   (*считывание и обработка дискретного сигнала с выбранного канала*)
   CASE #N_module OF
       4:  // Модуль 4
           CASE #N_chanel OF
               1:  #Signal := "Module4Chanel1";   //Канал 1
               2:  #Signal := "Module4Chanel2";   //Канал 2
               3:  #Signal := "Module4Chanel3";   //Канал 3
               4:  #Signal := "Module4Chanel4";   //Канал 4
               5:  #Signal := "Module4Chanel5";   //Канал 5
               6:  #Signal := "Module4Chanel6";   //Канал 6
               7:  #Signal := "Module4Chanel7";   //Канал 7
               8:  #Signal := "Module4Chanel8";   //Канал 8
               9:  #Signal := "Module4Chanel9";   //Канал 9
               10: #Signal := "Module4Chanel10";  //Канал 10
               11: #Signal := "Module4Chanel11";  //Канал 11
               12: #Signal := "Module4Chanel12";  //Канал 12
               13: #Signal := "Module4Chanel13";  //Канал 13
               14: #Signal := "Module4Chanel14";  //Канал 14
               15: #Signal := "Module4Chanel15";  //Канал 15
               16: #Signal := "Module4Chanel16";  //Канал 16
               ELSE
                   #Signal := FALSE;
           END_CASE;
       5:  // Модуль 5
           CASE #N_chanel OF
               1:  #Signal := "Module5Chanel1";   //Канал 1
               2:  #Signal := "Module5Chanel2";   //Канал 2
               3:  #Signal := "Module5Chanel3";   //Канал 3
               4:  #Signal := "Module5Chanel4";   //Канал 4
               5:  #Signal := "Module5Chanel5";   //Канал 5
               6:  #Signal := "Module5Chanel6";   //Канал 6
               7:  #Signal := "Module5Chanel7";   //Канал 7
               8:  #Signal := "Module5Chanel8";   //Канал 8
               9:  #Signal := "Module5Chanel9";   //Канал 9
               10: #Signal := "Module5Chanel10";  //Канал 10
               11: #Signal := "Module5Chanel11";  //Канал 11
               12: #Signal := "Module5Chanel12";  //Канал 12
               13: #Signal := "Module5Chanel13";  //Канал 13
               14: #Signal := "Module5Chanel14";  //Канал 14
               15: #Signal := "Module5Chanel15";  //Канал 15
               16: #Signal := "Module5Chanel16";  //Канал 16
               ELSE
                   #Signal := FALSE;
           END_CASE;
       6:  // Модуль 6
           CASE #N_chanel OF
               1:  #Signal := "Module6Chanel1";   //Канал 1
               2:  #Signal := "Module6Chanel2";   //Канал 2
               3:  #Signal := "Module6Chanel3";   //Канал 3
               4:  #Signal := "Module6Chanel4";   //Канал 4
               5:  #Signal := "Module6Chanel5";   //Канал 5
               6:  #Signal := "Module6Chanel6";   //Канал 6
               7:  #Signal := "Module6Chanel7";   //Канал 7
               8:  #Signal := "Module6Chanel8";   //Канал 8
               9:  #Signal := "Module6Chanel9";   //Канал 9
               10: #Signal := "Module6Chanel10";  //Канал 10
               11: #Signal := "Module6Chanel11";  //Канал 11
               12: #Signal := "Module6Chanel12";  //Канал 12
               13: #Signal := "Module6Chanel13";  //Канал 13
               14: #Signal := "Module6Chanel14";  //Канал 14
               15: #Signal := "Module6Chanel15";  //Канал 15
               16: #Signal := "Module6Chanel16";  //Канал 16
               ELSE
                   #Signal := FALSE;
           END_CASE;
       7:  // Модуль 7
           CASE #N_chanel OF
               1:  #Signal := "Module7Chanel1";   //Канал 1
               2:  #Signal := "Module7Chanel2";   //Канал 2
               3:  #Signal := "Module7Chanel3";   //Канал 3
               4:  #Signal := "Module7Chanel4";   //Канал 4
               5:  #Signal := "Module7Chanel5";   //Канал 5
               6:  #Signal := "Module7Chanel6";   //Канал 6
               7:  #Signal := "Module7Chanel7";   //Канал 7
               8:  #Signal := "Module7Chanel8";   //Канал 8
               9:  #Signal := "Module7Chanel9";   //Канал 9
               10: #Signal := "Module7Chanel10";  //Канал 10
               11: #Signal := "Module7Chanel11";  //Канал 11
               12: #Signal := "Module7Chanel12";  //Канал 12
               13: #Signal := "Module7Chanel13";  //Канал 13
               14: #Signal := "Module7Chanel14";  //Канал 14
               15: #Signal := "Module7Chanel15";  //Канал 15
               16: #Signal := "Module7Chanel16";  //Канал 16
               ELSE
                   #Signal := FALSE;
           END_CASE;
       8:  // Модуль 8
           CASE #N_chanel OF
               1:  #Signal := "Module8Chanel1";   //Канал 1
               2:  #Signal := "Module8Chanel2";   //Канал 2
               3:  #Signal := "Module8Chanel3";   //Канал 3
               4:  #Signal := "Module8Chanel4";   //Канал 4
               5:  #Signal := "Module8Chanel5";   //Канал 5
               6:  #Signal := "Module8Chanel6";   //Канал 6
               7:  #Signal := "Module8Chanel7";   //Канал 7
               8:  #Signal := "Module8Chanel8";   //Канал 8
               9:  #Signal := "Module8Chanel9";   //Канал 9
               10: #Signal := "Module8Chanel10";  //Канал 10
               11: #Signal := "Module8Chanel11";  //Канал 11
               12: #Signal := "Module8Chanel12";  //Канал 12
               13: #Signal := "Module8Chanel13";  //Канал 13
               14: #Signal := "Module8Chanel14";  //Канал 14
               15: #Signal := "Module8Chanel15";  //Канал 15
               16: #Signal := "Module8Chanel16";  //Канал 16
               ELSE
                   #Signal := FALSE;
           END_CASE;
       9:  // Модуль 9
           CASE #N_chanel OF
               1:  #Signal := "Module9Chanel1";   //Канал 1
               2:  #Signal := "Module9Chanel2";   //Канал 2
               3:  #Signal := "Module9Chanel3";   //Канал 3
               4:  #Signal := "Module9Chanel4";   //Канал 4
               5:  #Signal := "Module9Chanel5";   //Канал 5
               6:  #Signal := "Module9Chanel6";   //Канал 6
               7:  #Signal := "Module9Chanel7";   //Канал 7
               8:  #Signal := "Module9Chanel8";   //Канал 8
               9:  #Signal := "Module9Chanel9";   //Канал 9
               10: #Signal := "Module9Chanel10";  //Канал 10
               11: #Signal := "Module9Chanel11";  //Канал 11
               12: #Signal := "Module9Chanel12";  //Канал 12
               13: #Signal := "Module9Chanel13";  //Канал 13
               14: #Signal := "Module9Chanel14";  //Канал 14
               15: #Signal := "Module9Chanel15";  //Канал 15
               16: #Signal := "Module9Chanel16";  //Канал 16
               ELSE
                   #Signal := FALSE;
           END_CASE;
       ELSE
           #Signal := 0;
   END_CASE;
   IF NOT #Invert THEN
       #Value := #Signal;
   ELSE
       #Value := NOT #Signal;
   END_IF;
END_FUNCTION

FUNCTION "Write_outputs" : Void   // FC4, SCL
{ S7_Optimized_Access := 'TRUE' }
VERSION : 0.1
BEGIN
   (*ЗАПИСЬ ВЫХОДОВ*)
   (*Запись дискретных выходов*)
   (*ЗРГ команда «Больше»*)
   IF "Sensors".ZRG_control_open.Enable THEN
       "Write_discret_signal"(N_module := "Sensors".ZRG_control_open.N_module,
                              N_chanel := "Sensors".ZRG_control_open.N_chanel,
                              Value := "Sensors".ZRG_control_open.Value);
   END_IF;

   (*ЗРГ команда «Меньше»*)
   IF "Sensors".ZRG_control_close.Enable THEN
       "Write_discret_signal"(N_module := "Sensors".ZRG_control_close.N_module,
                              N_chanel := "Sensors".ZRG_control_close.N_chanel,
                              Value := "Sensors".ZRG_control_close.Value);
   END_IF;

   (*НАВ команда «Больше»*)
   IF "Sensors".NAV_control_open.Enable THEN
       "Write_discret_signal"(N_module := "Sensors".NAV_control_open.N_module,
                              N_chanel := "Sensors".NAV_control_open.N_chanel,
                              Value := "Sensors".NAV_control_open.Value);
   END_IF;

   (*НАВ команда «Меньше»*)
   IF "Sensors".NAV_control_close.Enable THEN
       "Write_discret_signal"(N_module := "Sensors".NAV_control_close.N_module,
                              N_chanel := "Sensors".NAV_control_close.N_chanel,
                              Value := "Sensors".NAV_control_close.Value);
   END_IF;

   (*НАД команда «Больше»*)
   IF "Sensors".NAD_control_open.Enable THEN
       "Write_discret_signal"(N_module := "Sensors".NAD_control_open.N_module,
                              N_chanel := "Sensors".NAD_control_open.N_chanel,
                              Value := "Sensors".NAD_control_open.Value);
   END_IF;

   (*НАД команда «Меньше»*)
   IF "Sensors".NAD_control_close.Enable THEN
       "Write_discret_signal"(N_module := "Sensors".NAD_control_close.N_module,
                              N_chanel := "Sensors".NAD_control_close.N_chanel,
                              Value := "Sensors".NAD_control_close.Value);
   END_IF;

   (*Индикация «Работа»*)
   IF "Sensors".Indication_RUN.Enable THEN
       "Write_discret_signal"(N_module := "Sensors".Indication_RUN.N_module,
                              N_chanel := "Sensors".Indication_RUN.N_chanel,
                              Value := "Sensors".Indication_RUN.Value);
   END_IF;

   (*Индикация «Авария»*)
   IF "Sensors".Indication_ALARM.Enable THEN
       "Write_discret_signal"(N_module := "Sensors".Indication_ALARM.N_module,
                              N_chanel := "Sensors".Indication_ALARM.N_chanel,
                              Value := "Sensors".Indication_ALARM.Value);
   END_IF;

   (*Индикация «Защиты в норме»*)
   IF "Sensors".Indication_NORMA.Enable THEN
       "Write_discret_signal"(N_module := "Sensors".Indication_NORMA.N_module,
                              N_chanel := "Sensors".Indication_NORMA.N_chanel,
                              Value := "Sensors".Indication_NORMA.Value);
   END_IF;

   (*Индикация «Готов к розжигу»*)
   IF "Sensors".Indication_READY.Enable THEN
       "Write_discret_signal"(N_module := "Sensors".Indication_READY.N_module,
                              N_chanel := "Sensors".Indication_READY.N_chanel,
                              Value := "Sensors".Indication_READY.Value);
   END_IF;

   (*ЗДГ команда «открыть»*)
   IF "Sensors".ZDG_control_open.Enable THEN
       "Write_discret_signal"(N_module := "Sensors".ZDG_control_open.N_module,
                              N_chanel := "Sensors".ZDG_control_open.N_chanel,
                              Value := "Sensors".ZDG_control_open.Value);
   END_IF;

   (*ЗДГ команда «закрыть»*)
   IF "Sensors".ZDG_control_close.Enable THEN
       "Write_discret_signal"(N_module := "Sensors".ZDG_control_close.N_module,
                              N_chanel := "Sensors".ZDG_control_close.N_chanel,
                              Value := "Sensors".ZDG_control_close.Value);
   END_IF;

   (*ЗДГ команда «стоп»*)
   IF "Sensors".ZDG_control_stop.Enable THEN
       "Write_discret_signal"(N_module := "Sensors".ZDG_control_stop.N_module,
                              N_chanel := "Sensors".ZDG_control_stop.N_chanel,
                              Value := "Sensors".ZDG_control_stop.Value);
   END_IF;

   (*ЗДГ команда «запрет открытия»*)
   IF "Sensors".ZDG_control_disable_open.Enable THEN
       "Write_discret_signal"(N_module := "Sensors".ZDG_control_disable_open.N_module,
                              N_chanel := "Sensors".ZDG_control_disable_open.N_chanel,
                              Value := "Sensors".ZDG_control_disable_open.Value);
   END_IF;

   (*КБ команда «закрыть»*)
   IF "Sensors".KB_control_close.Enable THEN
       "Write_discret_signal"(N_module := "Sensors".KB_control_close.N_module,
                              N_chanel := "Sensors".KB_control_close.N_chanel,
                              Value := "Sensors".KB_control_close.Value);
   END_IF;

   (*КО команда «открыть»*)
   IF "Sensors".KO_control_open.Enable THEN
       "Write_discret_signal"(N_module := "Sensors".KO_control_open.N_module,
                              N_chanel := "Sensors".KO_control_open.N_chanel,
                              Value := "Sensors".KO_control_open.Value);
   END_IF;

   (*КЗ команда «открыть»*)
   IF "Sensors".KZ_control_open.Enable THEN
       "Write_discret_signal"(N_module := "Sensors".KZ_control_open.N_module,
                              N_chanel := "Sensors".KZ_control_open.N_chanel,
                              Value := "Sensors".KZ_control_open.Value);
   END_IF;

   (*ИВН команда «включить»*)
   IF "Sensors".IVN_control_on.Enable THEN
       "Write_discret_signal"(N_module := "Sensors".IVN_control_on.N_module,
                              N_chanel := "Sensors".IVN_control_on.N_chanel,
                              Value := "Sensors".IVN_control_on.Value);
   END_IF;

   (*ПЗК1 команда «открыть»*)
   IF "Sensors".PZK1_control_open.Enable THEN
       "Write_discret_signal"(N_module := "Sensors".PZK1_control_open.N_module,
                              N_chanel := "Sensors".PZK1_control_open.N_chanel,
                              Value := "Sensors".PZK1_control_open.Value);
   END_IF;

   (*ПЗК2 команда «открыть»*)
   IF "Sensors".PZK2_control_open.Enable THEN
       "Write_discret_signal"(N_module := "Sensors".PZK2_control_open.N_module,
                              N_chanel := "Sensors".PZK2_control_open.N_chanel,
                              Value := "Sensors".PZK2_control_open.Value);
   END_IF;

   (*ЗДСВ перед котлом команда «открыть»*)
   IF "Sensors".ZDSV_before_boiler_control_open.Enable THEN
       "Write_discret_signal"(N_module := "Sensors".ZDSV_before_boiler_control_open.N_module,
                              N_chanel := "Sensors".ZDSV_before_boiler_control_open.N_chanel,
                              Value := "Sensors".ZDSV_before_boiler_control_open.Value);
   END_IF;

   (*ЗДСВ перед котлом команда «закрыть»*)
   IF "Sensors".ZDSV_before_boiler_control_close.Enable THEN
       "Write_discret_signal"(N_module := "Sensors".ZDSV_before_boiler_control_close.N_module,
                              N_chanel := "Sensors".ZDSV_before_boiler_control_close.N_chanel,
                              Value := "Sensors".ZDSV_before_boiler_control_close.Value);
   END_IF;

   (*ЗДСВ перед котлом команда «стоп»*)
   IF "Sensors".ZDSV_before_boiler_control_stop.Enable THEN
       "Write_discret_signal"(N_module := "Sensors".ZDSV_before_boiler_control_stop.N_module,
                              N_chanel := "Sensors".ZDSV_before_boiler_control_stop.N_chanel,
                              Value := "Sensors".ZDSV_before_boiler_control_stop.Value);
   END_IF;

   (*ЗДСВ перед котлом команда «разрешение на закрытие»*)
   IF "Sensors".ZDSV_before_boiler_control_disable_close.Enable THEN
       "Write_discret_signal"(N_module := "Sensors".ZDSV_before_boiler_control_disable_close.N_module,
                              N_chanel := "Sensors".ZDSV_before_boiler_control_disable_close.N_chanel,
                              Value := "Sensors".ZDSV_before_boiler_control_disable_close.Value);
   END_IF;

   (*ЗДСВ после котла команда «открыть»*)
   IF "Sensors".ZDSV_after_boiler_control_open.Enable THEN
       "Write_discret_signal"(N_module := "Sensors".ZDSV_after_boiler_control_open.N_module,
                              N_chanel := "Sensors".ZDSV_after_boiler_control_open.N_chanel,
                              Value := "Sensors".ZDSV_after_boiler_control_open.Value);
   END_IF;

   (*ЗДСВ после котла команда «закрыть»*)
   IF "Sensors".ZDSV_after_boiler_control_close.Enable THEN
       "Write_discret_signal"(N_module := "Sensors".ZDSV_after_boiler_control_close.N_module,
                              N_chanel := "Sensors".ZDSV_after_boiler_control_close.N_chanel,
                              Value := "Sensors".ZDSV_after_boiler_control_close.Value);
   END_IF;

   (*ЗДСВ после котла команда «стоп»*)
   IF "Sensors".ZDSV_after_boiler_control_stop.Enable THEN
       "Write_discret_signal"(N_module := "Sensors".ZDSV_after_boiler_control_stop.N_module,
                              N_chanel := "Sensors".ZDSV_after_boiler_control_stop.N_chanel,
                              Value := "Sensors".ZDSV_after_boiler_control_stop.Value);
   END_IF;

   (*ЗДСВ после котла команда «разрешение на закрытие»*)
   IF "Sensors".ZDSV_after_boiler_control_disable_close.Enable THEN
       "Write_discret_signal"(N_module := "Sensors".ZDSV_after_boiler_control_disable_close.N_module,
                              N_chanel := "Sensors".ZDSV_after_boiler_control_disable_close.N_chanel,
                              Value := "Sensors".ZDSV_after_boiler_control_disable_close.Value);
   END_IF;

   (*Включение аварийной сигнализации*)
   IF "Sensors".control_alarm_signal.Enable THEN
       "Write_discret_signal"(N_module := "Sensors".control_alarm_signal.N_module,
                              N_chanel := "Sensors".control_alarm_signal.N_chanel,
                              Value := "Sensors".control_alarm_signal.Value);
   END_IF;

   (*ДВ команда «пуск»*)
   IF "Sensors".DV_control_start.Enable THEN
       "Write_discret_signal"(N_module := "Sensors".DV_control_start.N_module,
                              N_chanel := "Sensors".DV_control_start.N_chanel,
                              Value := "Sensors".DV_control_start.Value);
   END_IF;

   (*ДВ команда «стоп»*)
   IF "Sensors".DV_control_stop.Enable THEN
       "Write_discret_signal"(N_module := "Sensors".DV_control_stop.N_module,
                              N_chanel := "Sensors".DV_control_stop.N_chanel,
                              Value := "Sensors".DV_control_stop.Value);
   END_IF;

   (*ДС команда «пуск»*)
   IF "Sensors".DS_control_start.Enable THEN
       "Write_discret_signal"(N_module := "Sensors".DS_control_start.N_module,
                              N_chanel := "Sensors".DS_control_start.N_chanel,
                              Value := "Sensors".DS_control_start.Value);
   END_IF;

   (*ДС команда «стоп»*)
   IF "Sensors".DS_control_stop.Enable THEN
       "Write_discret_signal"(N_module := "Sensors".DS_control_stop.N_module,
                              N_chanel := "Sensors".DS_control_stop.N_chanel,
                              Value := "Sensors".DS_control_stop.Value);
   END_IF;

   (*Запись аналоговых выходов*)
   (*Задание для ПЧ ДВ*)
   IF "Sensors".DV_control_frequency.Enable THEN
       "Write_analog_4_20"(N_module := "Sensors".DV_control_frequency.N_module,
                           N_chanel := "Sensors".DV_control_frequency.N_chanel,
                           Value := "Sensors".DV_control_frequency.Value,
                           Low_limit_phisical_current := "Sensors".DV_control_frequency.Low_limit_phisical_current,
                           High_limit_phisical_current := "Sensors".DV_control_frequency.High_limit_phisical_current,
                           Current_DAC => "Sensors".DV_control_frequency.Current_DAC);
       //применение изменений значений точек для пересчета сигнала
       IF "Sensors".DV_control_frequency.Apply THEN
           "Sensors".DV_control_frequency.Low_limit_phisical_current := "Sensors".DV_control_frequency.Low_limit_phisical_new;
           "Sensors".DV_control_frequency.High_limit_phisical_current := "Sensors".DV_control_frequency.High_limit_phisical_new;
           "Sensors".DV_control_frequency.Apply := false;
       END_IF;
   ELSE
       "Sensors".DV_control_frequency.Apply := false;
   END_IF;

   (*Задание для ПЧ ДС*)
   IF "Sensors".DS_control_frequency.Enable THEN
       "Write_analog_4_20"(N_module := "Sensors".DS_control_frequency.N_module,
                           N_chanel := "Sensors".DS_control_frequency.N_chanel,
                           Value := "Sensors".DS_control_frequency.Value,
                           Low_limit_phisical_current := "Sensors".DS_control_frequency.Low_limit_phisical_current,
                           High_limit_phisical_current := "Sensors".DS_control_frequency.High_limit_phisical_current,
                           Current_DAC => "Sensors".DS_control_frequency.Current_DAC);
       //применение изменений значений точек для пересчета сигнала
       IF "Sensors".DS_control_frequency.Apply THEN
           "Sensors".DS_control_frequency.Low_limit_phisical_current := "Sensors".DS_control_frequency.Low_limit_phisical_new;
           "Sensors".DS_control_frequency.High_limit_phisical_current := "Sensors".DS_control_frequency.High_limit_phisical_new;
           "Sensors".DS_control_frequency.Apply := false;
       END_IF;
   ELSE
       "Sensors".DS_control_frequency.Apply := false;
   END_IF;
END_FUNCTION

FUNCTION "Write_discret_signal" : Void   // FC5, SCL
{ S7_Optimized_Access := 'TRUE' }
VERSION : 0.1
   VAR_INPUT
      Value : Bool;   // Текущее значение сигнала
   END_VAR
   VAR_IN_OUT
      N_module : USInt;   // № модуля (начиная с 1)
      N_chanel : USInt;   // № канала (начиная с 1)
   END_VAR
BEGIN
   (*проверка правильности введеного значения № Модуля*)
   IF #N_module < 10 OR #N_module > 12 THEN
       #N_module := 0;
   END_IF;

   (*проверка правильности введеного значения № Канала*)
   IF #N_module = 0 THEN
       #N_chanel := 0;
   ELSE
       IF #N_chanel < 1 OR #N_chanel > 16 THEN
           #N_chanel := 0;
       END_IF;
   END_IF;

   (*запись дискретного сигнала в выбранный канал*)
   CASE #N_module OF
       10:  // Модуль 10
           CASE #N_chanel OF
               1:
                   "Module10Chanel1" := #Value;   //Канал 1
               2:
                   "Module10Chanel2" := #Value;   //Канал 2
               3:
                   "Module10Chanel3" := #Value;   //Канал 3
               4:
                   "Module10Chanel4" := #Value;   //Канал 4
               5:
                   "Module10Chanel5" := #Value;   //Канал 5
               6:
                   "Module10Chanel6" := #Value;   //Канал 6
               7:
                   "Module10Chanel7" := #Value;   //Канал 7
               8:
                   "Module10Chanel8" := #Value;   //Канал 8
               9:
                   "Module10Chanel9" := #Value;   //Канал 9
               10:
                   "Module10Chanel10" := #Value;   //Канал 10
               11:
                   "Module10Chanel11" := #Value;   //Канал 11
               12:
                   "Module10Chanel12" := #Value;   //Канал 12
               13:
                   "Module10Chanel13" := #Value;   //Канал 13
               14:
                   "Module10Chanel14" := #Value;   //Канал 14
               15:
                   "Module10Chanel15" := #Value;   //Канал 15
               16:
                   "Module10Chanel16" := #Value;   //Канал 16
           END_CASE;
       11:  // Модуль 11
           CASE #N_chanel OF
               1:
                   "Module11Chanel1" := #Value;   //Канал 1
               2:
                   "Module11Chanel2" := #Value;   //Канал 2
               3:
                   "Module11Chanel3" := #Value;   //Канал 3
               4:
                   "Module11Chanel4" := #Value;   //Канал 4
               5:
                   "Module11Chanel5" := #Value;   //Канал 5
               6:
                   "Module11Chanel6" := #Value;   //Канал 6
               7:
                   "Module11Chanel7" := #Value;   //Канал 7
               8:
                   "Module11Chanel8" := #Value;   //Канал 8
               9:
                   "Module11Chanel9" := #Value;   //Канал 9
               10:
                   "Module11Chanel10" := #Value;   //Канал 10
               11:
                   "Module11Chanel11" := #Value;   //Канал 11
               12:
                   "Module11Chanel12" := #Value;   //Канал 12
               13:
                   "Module11Chanel13" := #Value;   //Канал 13
               14:
                   "Module11Chanel14" := #Value;   //Канал 14
               15:
                   "Module11Chanel15" := #Value;   //Канал 15
               16:
                   "Module11Chanel16" := #Value;   //Канал 16
           END_CASE;
       12:  // Модуль 12
           CASE #N_chanel OF
               1:
                   "Module12Chanel1" := #Value;   //Канал 1
               2:
                   "Module12Chanel2" := #Value;   //Канал 2
               3:
                   "Module12Chanel3" := #Value;   //Канал 3
               4:
                   "Module12Chanel4" := #Value;   //Канал 4
               5:
                   "Module12Chanel5" := #Value;   //Канал 5
               6:
                   "Module12Chanel6" := #Value;   //Канал 6
               7:
                   "Module12Chanel7" := #Value;   //Канал 7
               8:
                   "Module12Chanel8" := #Value;   //Канал 8
               9:
                   "Module12Chanel9" := #Value;   //Канал 9
               10:
                   "Module12Chanel10" := #Value;   //Канал 10
               11:
                   "Module12Chanel11" := #Value;   //Канал 11
               12:
                   "Module12Chanel12" := #Value;   //Канал 12
               13:
                   "Module12Chanel13" := #Value;   //Канал 13
               14:
                   "Module12Chanel14" := #Value;   //Канал 14
               15:
                   "Module12Chanel15" := #Value;   //Канал 15
               16:
                   "Module12Chanel16" := #Value;   //Канал 16
           END_CASE;
   END_CASE;
END_FUNCTION

FUNCTION "Write_analog_4_20" : Void   // FC6, SCL
{ S7_Optimized_Access := 'TRUE' }
VERSION : 0.1
   VAR_INPUT
      Value : Real;   // Текущее значение в физической величине
      Low_limit_phisical_current : Real;   // Нижний предел датчика в физической величине текущий
      High_limit_phisical_current : Real;   // Верхний предел датчика в физической величине текущий
   END_VAR
   VAR_OUTPUT
      Current_DAC : Int;   // Текущий код ЦАП
   END_VAR
   VAR_IN_OUT
      N_module : USInt;   // № модуля (начиная с 13)
      N_chanel : USInt;   // № канала (начиная с 1)
   END_VAR
   VAR_TEMP
      DAC : Int;   // Текущий код ЦАП (для использования внутри функции)
   END_VAR
BEGIN
   (*проверка правильности введеного значения № Модуля*)
   IF #N_module < 13 OR #N_module > 13 THEN
       #N_module := 0;
   END_IF;

   (*проверка правильности введеного значения № Канала*)
   IF #N_module = 0 THEN
       #N_chanel := 0;
   ELSE
       IF #N_chanel < 1 OR #N_chanel > 4 THEN
           #N_chanel := 0;
       END_IF;
   END_IF;

   (*Вычисление кода ЦАП*)
   #DAC := REAL_TO_INT(((INT_TO_REAL(27648 - 0)) / (#High_limit_phisical_current - #Low_limit_phisical_current)) * #Value) + 0;
   #Current_DAC := #DAC;

   (*запись кода ЦАП в выбранной канал*)
   CASE #N_module OF
       13:  // Модуль 13
           CASE #N_chanel OF
               1:
                   "Module13Chanel1" := #DAC;   //Канал 1
               2:
                   "Module13Chanel2" := #DAC;   //Канал 2
               3:
                   "Module13Chanel3" := #DAC;   //Канал 3
               4:
                   "Module13Chanel4" := #DAC;   //Канал 4
           END_CASE;
   END_CASE;
END_FUNCTION

FUNCTION "Alarms" : Void   // FC7, SCL
{ S7_Optimized_Access := 'TRUE' }
VERSION : 0.1
BEGIN
   (*таймеры*)
   "TON_alarm_1_DB".TON(IN := "Timer".alarm_1_IN,
                        PT := "Timer".alarm_1_PT,
                        Q => "Timer".alarm_1_Q);
   "TON_alarm_2_DB".TON(IN := "Timer".alarm_2_IN,
                        PT := "Timer".alarm_2_PT,
                        Q => "Timer".alarm_2_Q);
   "TON_alarm_3_DB".TON(IN := "Timer".alarm_3_IN,
                        PT := "Timer".alarm_3_PT,
                        Q => "Timer".alarm_3_Q);
   "TON_alarm_4_DB".TON(IN := "Timer".alarm_4_IN,
                        PT := "Timer".alarm_4_PT,
                        Q => "Timer".alarm_4_Q);
   "TON_alarm_5_DB".TON(IN := "Timer".alarm_5_IN,
                        PT := "Timer".alarm_5_PT,
                        Q => "Timer".alarm_5_Q);
   "TON_alarm_6_DB".TON(IN := "Timer".alarm_6_IN,
                        PT := "Timer".alarm_6_PT,
                        Q => "Timer".alarm_6_Q);
   "TON_alarm_7_DB".TON(IN := "Timer".alarm_7_IN,
                        PT := "Timer".alarm_7_PT,
                        Q => "Timer".alarm_7_Q);
   "TON_alarm_8_DB".TON(IN := "Timer".alarm_8_IN,
                        PT := "Timer".alarm_8_PT,
                        Q => "Timer".alarm_8_Q);
   "TON_alarm_9_DB".TON(IN := "Timer".alarm_9_IN,
                        PT := "Timer".alarm_9_PT,
                        Q => "Timer".alarm_9_Q);
   "TON_alarm_10_DB".TON(IN := "Timer".alarm_10_IN,
                         PT := "Timer".alarm_10_PT,
                         Q => "Timer".alarm_10_Q);
   "TON_alarm_11_DB".TON(IN := "Timer".alarm_11_IN,
                         PT := "Timer".alarm_11_PT,
                         Q => "Timer".alarm_11_Q);
   "TON_alarm_12_DB".TON(IN := "Timer".alarm_12_IN,
                         PT := "Timer".alarm_12_PT,
                         Q => "Timer".alarm_12_Q);
   "TON_alarm_13_DB".TON(IN := "Timer".alarm_13_IN,
                         PT := "Timer".alarm_13_PT,
                         Q => "Timer".alarm_13_Q);
   "TON_alarm_14_DB".TON(IN := "Timer".alarm_14_IN,
                         PT := "Timer".alarm_14_PT,
                         Q => "Timer".alarm_14_Q);
   "TON_alarm_15_DB".TON(IN := "Timer".alarm_15_IN,
                         PT := "Timer".alarm_15_PT,
                         Q => "Timer".alarm_15_Q);
   "TON_alarm_16_DB".TON(IN := "Timer".alarm_16_IN,
                         PT := "Timer".alarm_16_PT,
                         Q => "Timer".alarm_16_Q);
   "TON_alarm_17_DB".TON(IN := "Timer".alarm_17_IN,
                         PT := "Timer".alarm_17_PT,
                         Q => "Timer".alarm_17_Q);

   "TON_warning_1_DB".TON(IN := "Timer".warning_1_IN,
                          PT := "Timer".warning_1_PT,
                          Q => "Timer".warning_1_Q);
   "TON_warning_2_DB".TON(IN := "Timer".warning_2_IN,
                          PT := "Timer".warning_2_PT,
                          Q => "Timer".warning_2_Q);

   "TON_test_sound_DB".TON(IN := "Timer".test_sound_IN,
                           PT := "Timer".test_sound_PT,
                           Q => "Timer".test_sound_Q);

   (*Формирование аварийных сообщений*)
   (*Повышение давления газа перед БГ*)
   "Timer".alarm_1_PT := T_CONV(INT_TO_DINT("Alarms_and_warnings".TIME_Alarm_P_gas_before_BG_max) * 1000);
   IF "Alarms_and_warnings".Enable_Alarm_P_gas_before_BG_max THEN
       "Timer".alarm_1_IN := "Sensors".P_gas_before_BG_max.Value OR ("Sensors".P_gas_before_BG.Value > "Alarms_and_warnings".SP_alarm_H_P_gas_before_BG AND NOT "Alarms_and_warnings".Warning_sensor_P_gas_before_BG AND "Sensors".P_gas_before_BG.Enable);
       IF "Timer".alarm_1_Q THEN
           "Alarms_and_warnings".Alarm_P_gas_before_BG_max := TRUE;
       END_IF;
   ELSE
       "Timer".alarm_1_IN := FALSE;
       //"Alarms_and_warnings".Alarm_P_gas_before_BG_max := FALSE;
   END_IF;
   (*Формирование технологической защиты. Повышение давления газа перед БГ*)
   IF NOT "Protections".BLOCK_P_gas_before_BG_max THEN
       "Protections".P_gas_before_BG_max := "Timer".alarm_1_Q;
   ELSE
       "Protections".P_gas_before_BG_max := FALSE;
   END_IF;

   (*Понижение давления газа перед БГ*)
   "Timer".alarm_2_PT := T_CONV(INT_TO_DINT("Alarms_and_warnings".TIME_Alarm_P_gas_before_BG_min) * 1000);
   IF "Alarms_and_warnings".Enable_Alarm_P_gas_before_BG_min THEN
       "Timer".alarm_2_IN := "Sensors".P_gas_before_BG_min.Value OR ("Sensors".P_gas_before_BG.Value < "Alarms_and_warnings".SP_alarm_L_P_gas_before_BG AND NOT "Alarms_and_warnings".Warning_sensor_P_gas_before_BG AND "Sensors".P_gas_before_BG.Enable);
       IF "Timer".alarm_2_Q THEN
           "Alarms_and_warnings".Alarm_P_gas_before_BG_min := TRUE;
       END_IF;
   ELSE
       "Timer".alarm_2_IN := FALSE;
       //"Alarms_and_warnings".Alarm_P_gas_before_BG_min := FALSE;
   END_IF;
   (*Формирование технологической защиты. Понижение давления газа перед БГ*)
   IF NOT "Protections".BLOCK_P_gas_before_BG_min THEN
       "Protections".P_gas_before_BG_min := "Timer".alarm_2_Q;
   ELSE
       "Protections".P_gas_before_BG_min := FALSE;
   END_IF;

   (*Понижение давления газа перед горелкой*)
   "Timer".alarm_3_PT := T_CONV(INT_TO_DINT("Alarms_and_warnings".TIME_Alarm_P_gas_before_burner_min) * 1000);
   IF "Alarms_and_warnings".Enable_Alarm_P_gas_before_burner_min THEN
       "Timer".alarm_3_IN := "Sensors".P_gas_before_burner_min.Value OR ("Sensors".P_gas_before_burner.Value < "Alarms_and_warnings".SP_alarm_L_P_gas_before_burner AND NOT "Alarms_and_warnings".Warning_sensor_P_gas_before_burner AND "Sensors".P_gas_before_burner.Enable);
       IF "Timer".alarm_3_Q THEN
           "Alarms_and_warnings".Alarm_P_gas_before_burner_min := TRUE;
       END_IF;
   ELSE
       "Timer".alarm_3_IN := FALSE;
       //"Alarms_and_warnings".Alarm_P_gas_before_burner_min := FALSE;
   END_IF;
   (*Формирование технологической защиты. Понижение давления газа перед горелкой*)
   IF NOT "Protections".BLOCK_P_gas_before_burner_min THEN
       "Protections".P_gas_before_burner_min := "Timer".alarm_3_Q;
   ELSE
       "Protections".P_gas_before_burner_min := FALSE;
   END_IF;

   (*Повышение давления газа перед горелкой*)
   "Timer".alarm_4_PT := T_CONV(INT_TO_DINT("Alarms_and_warnings".TIME_Alarm_P_gas_before_burner_max) * 1000);
   IF "Alarms_and_warnings".Enable_Alarm_P_gas_before_burner_max THEN
       "Timer".alarm_4_IN := "Sensors".P_gas_before_burner_max.Value OR ("Sensors".P_gas_before_burner.Value > "Alarms_and_warnings".SP_alarm_H_P_gas_before_burner AND NOT "Alarms_and_warnings".Warning_sensor_P_gas_before_burner AND "Sensors".P_gas_before_burner.Enable);
       IF "Timer".alarm_4_Q THEN
           "Alarms_and_warnings".Alarm_P_gas_before_burner_max := TRUE;
       END_IF;
   ELSE
       "Timer".alarm_4_IN := FALSE;
       //"Alarms_and_warnings".Alarm_P_gas_before_burner_max := FALSE;
   END_IF;
   (*Формирование технологической защиты. Повышение давления газа перед горелкой*)
   IF NOT "Protections".BLOCK_P_gas_before_burner_max THEN
       "Protections".P_gas_before_burner_max := "Timer".alarm_4_Q;
   ELSE
       "Protections".P_gas_before_burner_max := FALSE;
   END_IF;

   (*Отключение ДС*)
   "Timer".alarm_5_PT := T_CONV(INT_TO_DINT("Alarms_and_warnings".TIME_Alarm_DS_off) * 1000);
   IF "Alarms_and_warnings".Enable_Alarm_DS_off THEN
       "Timer".alarm_5_IN := (NOT "Sensors".DS_invertor_on.Value AND NOT "Sensors".DS_powergrid_on.Value);
       IF "Timer".alarm_5_Q THEN
           "Alarms_and_warnings".Alarm_DS_off := TRUE;
       END_IF;
   ELSE
       "Timer".alarm_5_IN := FALSE;
       //"Alarms_and_warnings".Alarm_DS_off := FALSE;
   END_IF;
   (*Формирование технологической защиты. Отключение ДС*)
   IF NOT "Protections".BLOCK_DS_off THEN
       "Protections".DS_off := "Timer".alarm_5_Q;
   ELSE
       "Protections".DS_off := FALSE;
   END_IF;

   (*Отключение ДВ*)
   "Timer".alarm_6_PT := T_CONV(INT_TO_DINT("Alarms_and_warnings".TIME_Alarm_DV_off) * 1000);
   IF "Alarms_and_warnings".Enable_Alarm_DV_off THEN
       "Timer".alarm_6_IN := (NOT "Sensors".DV_invertor_on.Value AND NOT "Sensors".DV_powergrid_on.Value);
       IF "Timer".alarm_6_Q THEN
           "Alarms_and_warnings".Alarm_DV_off := TRUE;
       END_IF;
   ELSE
       "Timer".alarm_6_IN := FALSE;
       //"Alarms_and_warnings".Alarm_DV_off := FALSE;
   END_IF;
   (*Формирование технологической защиты. Отключение ДВ*)
   IF NOT "Protections".BLOCK_DV_off THEN
       "Protections".DV_off := "Timer".alarm_6_Q;
   ELSE
       "Protections".DV_off := FALSE;
   END_IF;

   (*Понижение разряжения в топке*)
   "Timer".alarm_7_PT := T_CONV(INT_TO_DINT("Alarms_and_warnings".TIME_Alarm_dP_furnace_boiler_min) * 1000);
   IF "Alarms_and_warnings".Enable_Alarm_dP_furnace_boiler_min THEN
       "Timer".alarm_7_IN := "Sensors".dP_furnace_boiler_min.Value OR ("Sensors".dP_furnace_boiler.Value > "Alarms_and_warnings".SP_alarm_L_dP_furnace_boiler AND NOT "Alarms_and_warnings".Warning_sensor_dP_furnace_boiler AND "Sensors".dP_furnace_boiler.Enable);
       IF "Timer".alarm_7_Q THEN
           "Alarms_and_warnings".Alarm_dP_furnace_boiler_min := TRUE;
       END_IF;
   ELSE
       "Timer".alarm_7_IN := FALSE;
       //"Alarms_and_warnings".Alarm_dP_furnace_boiler_min := FALSE;
   END_IF;
   (*Формирование технологической защиты. Понижение разряжения в топке*)
   IF NOT "Protections".BLOCK_dP_in_furnance_min THEN
       "Protections".dP_in_furnance_min := "Timer".alarm_7_Q;
   ELSE
       "Protections".dP_in_furnance_min := FALSE;
   END_IF;

   (*Понижение давления воздуха перед горелкой *)
   "Timer".alarm_8_PT := T_CONV(INT_TO_DINT("Alarms_and_warnings".TIME_Alarm_P_air_before_burner_min) * 1000);
   IF "Alarms_and_warnings".Enable_Alarm_P_air_before_burner_min THEN
       "Timer".alarm_8_IN := "Sensors".P_air_before_burner_min.Value OR ("Sensors".P_air_burner.Value < "Alarms_and_warnings".SP_alarm_L_P_air_before_burner AND NOT "Alarms_and_warnings".Warning_sensor_P_air_burner AND "Sensors".P_air_burner.Enable);
       IF "Timer".alarm_8_Q THEN
           "Alarms_and_warnings".Alarm_P_air_before_burner_min := TRUE;
       END_IF;
   ELSE
       "Timer".alarm_8_IN := FALSE;
       //"Alarms_and_warnings".Alarm_P_air_before_burner_min := FALSE;
   END_IF;
   (*Формирование технологической защиты. Понижение давления воздуха перед горелкой*)
   IF NOT "Protections".BLOCK_P_air_before_burner_min THEN
       "Protections".P_air_before_burner_min := "Timer".alarm_8_Q;
   ELSE
       "Protections".P_air_before_burner_min := FALSE;
   END_IF;

   (*Понижение давления сетевой воды за котлом*)
   "Timer".alarm_9_PT := T_CONV(INT_TO_DINT("Alarms_and_warnings".TIME_Alarm_P_water_after_boiler_min) * 1000);
   IF "Alarms_and_warnings".Enable_Alarm_P_water_after_boiler_min THEN
       "Timer".alarm_9_IN := "Sensors".P_water_after_boiler_min.Value OR ("Sensors".P_water_after_boiler.Value < "Alarms_and_warnings".SP_alarm_L_P_water_after_boiler AND NOT "Alarms_and_warnings".Warning_sensor_P_water_after_boiler AND "Sensors".P_water_after_boiler.Enable);
       IF "Timer".alarm_9_Q THEN
           "Alarms_and_warnings".Alarm_P_water_after_boiler_min := TRUE;
       END_IF;
   ELSE
       "Timer".alarm_9_IN := FALSE;
       //"Alarms_and_warnings".Alarm_P_water_after_boiler_min := FALSE;
   END_IF;
   (*Формирование технологической защиты. Понижение давления сетевой воды за котлом*)
   IF NOT "Protections".BLOCK_P_water_after_boiler_min THEN
       "Protections".P_water_after_boiler_min := "Timer".alarm_9_Q;
   ELSE
       "Protections".P_water_after_boiler_min := FALSE;
   END_IF;

   (*Повышение давления сетевой воды за котлом*)
   "Timer".alarm_10_PT := T_CONV(INT_TO_DINT("Alarms_and_warnings".TIME_Alarm_P_water_after_boiler_max) * 1000);
   IF "Alarms_and_warnings".Enable_Alarm_P_water_after_boiler_max THEN
       "Timer".alarm_10_IN := "Sensors".P_water_after_boiler_max.Value OR ("Sensors".P_water_after_boiler.Value > "Alarms_and_warnings".SP_alarm_H_P_water_after_boiler AND NOT "Alarms_and_warnings".Warning_sensor_P_water_after_boiler AND "Sensors".P_water_after_boiler.Enable);
       IF "Timer".alarm_10_Q THEN
           "Alarms_and_warnings".Alarm_P_water_after_boiler_max := TRUE;
       END_IF;
   ELSE
       "Timer".alarm_10_IN := FALSE;
       //"Alarms_and_warnings".Alarm_P_water_after_boiler_max := FALSE;
   END_IF;
   (*Формирование технологической защиты. Повышение давления сетевой воды за котлом*)
   IF NOT "Protections".BLOCK_P_water_after_boiler_max THEN
       "Protections".P_water_after_boiler_max := "Timer".alarm_10_Q;
   ELSE
       "Protections".P_water_after_boiler_max := FALSE;
   END_IF;

   (*Повышение температуры сетевой воды за котлом*)
   "Timer".alarm_11_PT := T_CONV(INT_TO_DINT("Alarms_and_warnings".TIME_Alarm_T_water_after_boiler_max) * 1000);
   IF "Alarms_and_warnings".Enable_Alarm_T_water_after_boiler_max THEN
       "Timer".alarm_11_IN := "Sensors".T_water_after_boiler_max.Value OR ("Sensors".T_water_after_boiler.Value > "Alarms_and_warnings".SP_alarm_H_T_water_after_boiler AND NOT "Alarms_and_warnings".Warning_sensor_T_water_after_boiler AND "Sensors".T_water_after_boiler.Enable);
       IF "Timer".alarm_11_Q THEN
           "Alarms_and_warnings".Alarm_T_water_after_boiler_max := TRUE;
       END_IF;
   ELSE
       "Timer".alarm_11_IN := FALSE;
       //"Alarms_and_warnings".Alarm_T_water_after_boiler_max := FALSE;
   END_IF;
   (*Формирование технологической защиты. Повышение температуры сетевой воды за котлом*)
   IF NOT "Protections".BLOCK_T_water_after_boiler_max THEN
       "Protections".T_water_after_boiler_max := "Timer".alarm_11_Q;
   ELSE
       "Protections".T_water_after_boiler_max := FALSE;
   END_IF;

   (*Понижение расхода сетевой воды через котел*)
   "Timer".alarm_12_PT := T_CONV(INT_TO_DINT("Alarms_and_warnings".TIME_Alarm_Q_water_boiler_min) * 1000);
   IF "Alarms_and_warnings".Enable_Alarm_Q_water_boiler_min THEN
       "Timer".alarm_12_IN := "Sensors".Q_water_boiler_min.Value OR ("Sensors".Q_water_boiler.Value < "Alarms_and_warnings".SP_alarm_L_Q_water_boiler AND "Sensors".Q_water_boiler.Enable);
       IF "Timer".alarm_12_Q THEN
           "Alarms_and_warnings".Alarm_Q_water_boiler_min := TRUE;
       END_IF;
   ELSE
       "Timer".alarm_12_IN := FALSE;
       //"Alarms_and_warnings".Alarm_Q_water_boiler_min := FALSE;
   END_IF;
   (*Формирование технологической защиты. Понижение расхода сетевой воды через котел*)
   IF NOT "Protections".BLOCK_Q_water_boiler_min THEN
       "Protections".Q_water_boiler_min := "Timer".alarm_12_Q;
   ELSE
       "Protections".Q_water_boiler_min := FALSE;
   END_IF;

   (*Невоспламенение или погасание факела горелки котла*)
   "Timer".alarm_13_PT := T_CONV(INT_TO_DINT("Alarms_and_warnings".TIME_Alarm_Not_flame_burner));
   IF "Alarms_and_warnings".Enable_Alarm_Not_flame_burner THEN
       "Timer".alarm_13_IN := NOT "Sensors".Burner_flame.Value;
       IF "Timer".alarm_13_Q THEN
           "Alarms_and_warnings".Alarm_Not_flame_burner := TRUE;
       END_IF;
   ELSE
       "Timer".alarm_13_IN := FALSE;
       //"Alarms_and_warnings".Alarm_Not_flame_burner := FALSE;
   END_IF;
   (*Формирование технологической защиты. Невоспламенение или погасание факела горелки котла*)
   IF NOT "Protections".BLOCK_Not_flame_burner THEN
       "Protections".Not_flame_burner := "Timer".alarm_13_Q;
   ELSE
       "Protections".Not_flame_burner := FALSE;
   END_IF;

   (*Нажата кнопка аварийного останова на панели оператора*)
   IF "Alarms_and_warnings".Enable_Alarm_stop_HMI THEN
       IF "FRONT_Btn_Alarm_stop_HMI" THEN
           "Alarms_and_warnings".Alarm_stop_HMI := TRUE;
       END_IF;
   ELSE
       ;
       //"Alarms_and_warnings".Alarm_stop_HMI := FALSE;
   END_IF;
   (*Формирование технологической защиты. Нажата кнопка аварийного останова на панели операторора*)
   IF NOT "Protections".BLOCK_Alarm_stop_HMI THEN
       "Protections".Alarm_stop_HMI := "FRONT_Btn_Alarm_stop_HMI";
   ELSE
       "Protections".Alarm_stop_HMI := FALSE;
   END_IF;

   (*Нажата кнопка аварийного останова на SCADA*)
   IF "Alarms_and_warnings".Enable_Alarm_stop_SCADA THEN
       IF "FRONT_Btn_Alarm_stop_SCADA" THEN
           "Alarms_and_warnings".Alarm_stop_SCADA := TRUE;
       END_IF;
   ELSE
       ;
       //"Alarms_and_warnings".Alarm_stop_SCADA := FALSE;
   END_IF;
   (*Формирование технологической защиты. Нажата кнопка аварийного останова на SCADA*)
   IF NOT "Protections".BLOCK_Alarm_stop_SCADA THEN
       "Protections".Alarm_stop_SCADA := "FRONT_Btn_Alarm_stop_SCADA";
   ELSE
       "Protections".Alarm_stop_SCADA := FALSE;
   END_IF;

   (*СО2 порог 2*)
   "Timer".alarm_14_PT := T_CONV(INT_TO_DINT("Alarms_and_warnings".TIME_Alarm_CO2_porog2));
   IF "Alarms_and_warnings".Enable_Alarm_CO2_porog2 THEN
       "Timer".alarm_14_IN := "Sensors".CO_2.Value;
       IF "Timer".alarm_14_Q THEN
           "Alarms_and_warnings".Alarm_CO2_porog2 := TRUE;
       END_IF;
   ELSE
       "Timer".alarm_14_IN := FALSE;
       //"Alarms_and_warnings".Alarm_CO2_porog2 := FALSE;
   END_IF;
   (*Формирование технологической защиты. СО2 порог 2*)
   "Protections".CO2_porog2 := FALSE;
   (*IF NOT "Protections".BLOCK_CO2_porog2 THEN
       "Protections".CO2_porog2 := "Alarms_and_warnings".Alarm_CO2_porog2;
   ELSE
       "Protections".CO2_porog2 := FALSE;
   END_IF;*)

   (*CH4*)
   "Timer".alarm_15_PT := T_CONV(INT_TO_DINT("Alarms_and_warnings".TIME_Alarm_CH4));
   IF "Alarms_and_warnings".Enable_Alarm_CH4 THEN
       "Timer".alarm_15_IN := "Sensors".CH4.Value;
       IF "Timer".alarm_15_Q THEN
           "Alarms_and_warnings".Alarm_CH4 := TRUE;
       END_IF;
   ELSE
       "Timer".alarm_15_IN := FALSE;
       //"Alarms_and_warnings".Alarm_CH4 := FALSE;
   END_IF;
   (*Формирование технологической защиты. CH4*)
   "Protections".CH4 := FALSE;
   (*IF NOT "Protections".BLOCK_CH4 THEN
       "Protections".CH4 := "Alarms_and_warnings".Alarm_CH4;
   ELSE
       "Protections".CH4 := FALSE;
   END_IF;*)

   (*Формирование предупредительных сообщений*)
   (*Предупреждение. Неисправность датчика T сетевой воды перед котлом*)
   IF "Sensors".T_water_before_boiler.Enable THEN
       "Alarms_and_warnings".Warning_sensor_T_water_before_boiler := "Sensors".T_water_before_boiler.Alarm_sensor;
   ELSE
       "Alarms_and_warnings".Warning_sensor_T_water_before_boiler := FALSE;
   END_IF;

   (*Предупреждение. Неисправность датчика P сетевой воды перед котлом*)
   IF "Sensors".P_water_before_boiler.Enable THEN
       "Alarms_and_warnings".Warning_sensor_P_water_before_boiler := "Sensors".P_water_before_boiler.Alarm_sensor;
   ELSE
       "Alarms_and_warnings".Warning_sensor_P_water_before_boiler := FALSE;
   END_IF;

   (*Предупреждение. Неисправность датчика dP сетевой воды через котел*)
   IF "Sensors".dP_water_boiler.Enable THEN
       "Alarms_and_warnings".Warning_sensor_dP_water_boiler := "Sensors".dP_water_boiler.Alarm_sensor;
   ELSE
       "Alarms_and_warnings".Warning_sensor_dP_water_boiler := FALSE;
   END_IF;

   (*Предупреждение. Неисправность датчика Т сетевой воды после котла*)
   IF "Sensors".T_water_after_boiler.Enable THEN
       "Alarms_and_warnings".Warning_sensor_T_water_after_boiler := "Sensors".T_water_after_boiler.Alarm_sensor;
   ELSE
       "Alarms_and_warnings".Warning_sensor_T_water_after_boiler := FALSE;
   END_IF;

   (*Предупреждение. Неисправность датчика P сетевой воды после котла*)
   IF "Sensors".P_water_after_boiler.Enable THEN
       "Alarms_and_warnings".Warning_sensor_P_water_after_boiler := "Sensors".P_water_after_boiler.Alarm_sensor;
   ELSE
       "Alarms_and_warnings".Warning_sensor_P_water_after_boiler := FALSE;
   END_IF;

   (*Предупреждение. Неисправность датчика dP сетевой воды через котел*)
   IF "Sensors".dP_water_boiler_1.Enable THEN
       "Alarms_and_warnings".Warning_sensor_dP_water_boiler_1 := "Sensors".dP_water_boiler_1.Alarm_sensor;
   ELSE
       "Alarms_and_warnings".Warning_sensor_dP_water_boiler_1 := FALSE;
   END_IF;

   (*Предупреждение. Неисправность датчика P сетевой воды перед котлом*)
   IF "Sensors".P_water_before_boiler_1.Enable THEN
       "Alarms_and_warnings".Warning_sensor_P_water_before_boiler_1 := "Sensors".P_water_before_boiler_1.Alarm_sensor;
   ELSE
       "Alarms_and_warnings".Warning_sensor_P_water_before_boiler_1 := FALSE;
   END_IF;

   (*Предупреждение. Неисправность датчика dP газа на котел*)
   IF "Sensors".dP_gas_boiler.Enable THEN
       "Alarms_and_warnings".Warning_sensor_dP_gas_boiler := "Sensors".dP_gas_boiler.Alarm_sensor;
   ELSE
       "Alarms_and_warnings".Warning_sensor_dP_gas_boiler := FALSE;
   END_IF;

   (*Предупреждение. Неисправность датчика разрежения в топке котла*)
   IF "Sensors".dP_furnace_boiler.Enable THEN
       "Alarms_and_warnings".Warning_sensor_dP_furnace_boiler := "Sensors".dP_furnace_boiler.Alarm_sensor;
   ELSE
       "Alarms_and_warnings".Warning_sensor_dP_furnace_boiler := FALSE;
   END_IF;

   (*Предупреждение. Неисправность датчика P газа между ПЗК-1 и ПЗК-2*)
   IF "Sensors".P_gas_before_PZK1_and_PZK2.Enable THEN
       "Alarms_and_warnings".Warning_sensor_P_gas_before_PZK1_and_PZK2 := "Sensors".P_gas_before_PZK1_and_PZK2.Alarm_sensor;
   ELSE
       "Alarms_and_warnings".Warning_sensor_P_gas_before_PZK1_and_PZK2 := FALSE;
   END_IF;

   (*Предупреждение. Неисправность датчика P газа перед горелкой*)
   IF "Sensors".P_gas_before_burner.Enable THEN
       "Alarms_and_warnings".Warning_sensor_P_gas_before_burner := "Sensors".P_gas_before_burner.Alarm_sensor;
   ELSE
       "Alarms_and_warnings".Warning_sensor_P_gas_before_burner := FALSE;
   END_IF;

   (*Предупреждение. Неисправность датчика P воздуха к горелке*)
   IF "Sensors".P_air_burner.Enable THEN
       "Alarms_and_warnings".Warning_sensor_P_air_burner := "Sensors".P_air_burner.Alarm_sensor;
   ELSE
       "Alarms_and_warnings".Warning_sensor_P_air_burner := FALSE;
   END_IF;

   (*Предупреждение. Неисправность датчика T уходящих газов*)
   IF "Sensors".T_exhaust_gas.Enable THEN
       "Alarms_and_warnings".Warning_sensor_T_exhaust_gas := "Sensors".T_exhaust_gas.Alarm_sensor;
   ELSE
       "Alarms_and_warnings".Warning_sensor_T_exhaust_gas := FALSE;
   END_IF;

   (*Предупреждение. Неисправность датчика положения рег. заслонки газа перед котлом*)
   IF "Sensors".ZRG_position.Enable THEN
       "Alarms_and_warnings".Warning_sensor_ZRG_position := "Sensors".ZRG_position.Alarm_sensor;
   ELSE
       "Alarms_and_warnings".Warning_sensor_ZRG_position := FALSE;
   END_IF;

   (*Предупреждение. Неисправность датчика положения направл. аппарата вентилятора*)
   IF "Sensors".NAV_position.Enable THEN
       "Alarms_and_warnings".Warning_sensor_NAV_position := "Sensors".NAV_position.Alarm_sensor;
   ELSE
       "Alarms_and_warnings".Warning_sensor_NAV_position := FALSE;
   END_IF;

   (*Предупреждение. Неисправность датчика положения направл. аппарата дымососа*)
   IF "Sensors".NAD_position.Enable THEN
       "Alarms_and_warnings".Warning_sensor_NAD_position := "Sensors".NAD_position.Alarm_sensor;
   ELSE
       "Alarms_and_warnings".Warning_sensor_NAD_position := FALSE;
   END_IF;

   (*Предупреждение. Неисправность датчика Текущ. значение ПЧ ДВ*)
   IF "Sensors".DV_current_frequency.Enable THEN
       "Alarms_and_warnings".Warning_sensor_DV_current_frequency := "Sensors".DV_current_frequency.Alarm_sensor;
   ELSE
       "Alarms_and_warnings".Warning_sensor_DV_current_frequency := FALSE;
   END_IF;

   (*Предупреждение. Неисправность датчика Текущ. значение ПЧ ДС*)
   IF "Sensors".DS_current_frequency.Enable THEN
       "Alarms_and_warnings".Warning_sensor_DS_current_frequency := "Sensors".DS_current_frequency.Alarm_sensor;
   ELSE
       "Alarms_and_warnings".Warning_sensor_DS_current_frequency := FALSE;
   END_IF;

   (*Предупреждение. Сработал ограничитель крутящего момента ЗДСВ перед котлом*)
   IF "Sensors".ZDSV_before_boiler_limit_rotational_moment.Enable THEN
       "Alarms_and_warnings".Warning_ZDSV_before_boiler_limit_rotational_moment := "Sensors".ZDSV_before_boiler_limit_rotational_moment.Value;
   ELSE
       "Alarms_and_warnings".Warning_ZDSV_before_boiler_limit_rotational_moment := FALSE;
   END_IF;

   (*Предупреждение. Сработал ограничитель крутящего момента ЗДСВ после котла*)
   IF "Sensors".ZDSV_after_boiler_limit_rotational_moment.Enable THEN
       "Alarms_and_warnings".Warning_ZDSV_after_boiler_limit_rotational_moment := "Sensors".ZDSV_after_boiler_limit_rotational_moment.Value;
   ELSE
       "Alarms_and_warnings".Warning_ZDSV_after_boiler_limit_rotational_moment := FALSE;
   END_IF;

   (*Предупреждение. Вызов к шакафу электропитания*)
   IF "Sensors".Call_power_supply_сabinet.Enable THEN
       "Alarms_and_warnings".Warning_сall_power_supply_сabinet := "Sensors".Call_power_supply_сabinet.Value;
   ELSE
       "Alarms_and_warnings".Warning_сall_power_supply_сabinet := FALSE;
   END_IF;

   (*Предупреждение. ДВ. Необходимо включить QF ПЧ*)
   IF "Sensors".DV_dist_control.Value AND "Sensors".DV_invertor_mode.Value AND NOT "Sensors".DV_invertor_QF_on.Value AND "Sensors".DV_invertor_QF_on.Enable THEN
       "Alarms_and_warnings".Warning_DV_need_on_QF_invertor := TRUE;
   ELSE
       "Alarms_and_warnings".Warning_DV_need_on_QF_invertor := FALSE;
   END_IF;

   (*Предупреждение. ДВ. Необходимо включить QF Сети*)
   IF "Sensors".DV_dist_control.Value AND "Sensors".DV_powergrid_mode.Value AND NOT "Sensors".DV_powergrid_QF_on.Value AND "Sensors".DV_powergrid_QF_on.Enable THEN
       "Alarms_and_warnings".Warning_DV_need_on_QF_powergrid := TRUE;
   ELSE
       "Alarms_and_warnings".Warning_DV_need_on_QF_powergrid := FALSE;
   END_IF;

   (*Предупреждение. ДВ. Неисправность напряжения в Сети ШУД*)
   IF "Sensors".DV_no_voltage.Enable THEN
       "Alarms_and_warnings".Warning_DV_no_voltage := "Sensors".DV_no_voltage.Value;
   ELSE
       "Alarms_and_warnings".Warning_DV_no_voltage := FALSE;
   END_IF;

   (*Предупреждение. ДС. Необходимо включить QF ПЧ*)
   IF "Sensors".DS_dist_control.Value AND "Sensors".DS_invertor_mode.Value AND NOT "Sensors".DS_invertor_QF_on.Value AND "Sensors".DS_invertor_QF_on.Enable THEN
       "Alarms_and_warnings".Warning_DS_need_on_QF_invertor := TRUE;
   ELSE
       "Alarms_and_warnings".Warning_DS_need_on_QF_invertor := FALSE;
   END_IF;

   (*Предупреждение. ДС. Необходимо включить QF Сети*)
   IF "Sensors".DS_dist_control.Value AND "Sensors".DS_powergrid_mode.Value AND NOT "Sensors".DS_powergrid_QF_on.Value AND "Sensors".DS_powergrid_QF_on.Enable THEN
       "Alarms_and_warnings".Warning_DS_need_on_QF_powergrid := TRUE;
   ELSE
       "Alarms_and_warnings".Warning_DS_need_on_QF_powergrid := FALSE;
   END_IF;

   (*Предупреждение. ДС. Неисправность напряжения в Сети ШУД*)
   IF "Sensors".DS_no_voltage.Enable THEN
       "Alarms_and_warnings".Warning_DS_no_voltage := "Sensors".DS_no_voltage.Value;
   ELSE
       "Alarms_and_warnings".Warning_DS_no_voltage := FALSE;
   END_IF;

   (*Предупреждение. Нет питания ШЭУ*)
   IF "Sensors".SHEU_voltage_ok.Enable THEN
       "Alarms_and_warnings".Warning_SHEU_no_voltage := NOT "Sensors".SHEU_voltage_ok.Value;
   ELSE
       "Alarms_and_warnings".Warning_SHEU_no_voltage := FALSE;
   END_IF;

   (*Предупреждение. Питание контроллера от ИБП*)
   IF "Sensors".Power_PLC_from_UPS.Enable THEN
       "Alarms_and_warnings".Warning_power_PLC_from_UPS := "Sensors".Power_PLC_from_UPS.Value;
   ELSE
       "Alarms_and_warnings".Warning_power_PLC_from_UPS := FALSE;
   END_IF;

   (*Предупреждение. Низкий заряд батареи ИБП*)
   IF "Sensors".UPS_Low_charge.Enable THEN
       "Alarms_and_warnings".Warning_UPS_Low_charge := "Sensors".UPS_Low_charge.Value;
   ELSE
       "Alarms_and_warnings".Warning_UPS_Low_charge := FALSE;
   END_IF;

   (*Предупреждение. Нет питания ЗРГ*)
   IF "Sensors".ZRG_voltage_ok.Enable THEN
       "Alarms_and_warnings".Warning_ZRG_no_voltage := NOT "Sensors".ZRG_voltage_ok.Value;
   ELSE
       "Alarms_and_warnings".Warning_ZRG_no_voltage := FALSE;
   END_IF;

   (*Предупреждение. Нет питания ЗДГ*)
   IF "Sensors".ZDG_voltage_ok.Enable THEN
       "Alarms_and_warnings".Warning_ZDG_no_voltage := NOT "Sensors".ZDG_voltage_ok.Value;
   ELSE
       "Alarms_and_warnings".Warning_ZDG_no_voltage := FALSE;
   END_IF;

   (*Предупреждение. Нет питания НАВ*)
   IF "Sensors".NAV_voltage_ok.Enable THEN
       "Alarms_and_warnings".Warning_NAV_no_voltage := NOT "Sensors".NAV_voltage_ok.Value;
   ELSE
       "Alarms_and_warnings".Warning_NAV_no_voltage := FALSE;
   END_IF;

   (*Предупреждение. Нет питания НАД*)
   IF "Sensors".NAD_voltage_ok.Enable THEN
       "Alarms_and_warnings".Warning_NAD_no_voltage := NOT "Sensors".NAD_voltage_ok.Value;
   ELSE
       "Alarms_and_warnings".Warning_NAD_no_voltage := FALSE;
   END_IF;

   (*Предупреждение. Нет питания ЗДСВ перед котлом*)
   IF "Sensors".ZDSV_before_boiler_voltage_ok.Enable THEN
       "Alarms_and_warnings".Warning_ZDSV_before_boiler_no_voltage := NOT "Sensors".ZDSV_before_boiler_voltage_ok.Value;
   ELSE
       "Alarms_and_warnings".Warning_ZDSV_before_boiler_no_voltage := FALSE;
   END_IF;

   (*Предупреждение. Нет питания ЗДСВ после котла*)
   IF "Sensors".ZDSV_after_boiler_voltage_ok.Enable THEN
       "Alarms_and_warnings".Warning_ZDSV_after_boiler_no_voltage := NOT "Sensors".ZDSV_after_boiler_voltage_ok.Value;
   ELSE
       "Alarms_and_warnings".Warning_ZDSV_after_boiler_no_voltage := FALSE;
   END_IF;

   (*Предупреждение. Авария ПЧ ДВ*)
   IF "Sensors".DV_Invertor_alarm.Enable AND "Sensors".DV_invertor_mode.Value THEN
       "Alarms_and_warnings".Warning_DV_invertor_alarm := "Sensors".DV_Invertor_alarm.Value;
   ELSE
       "Alarms_and_warnings".Warning_DV_invertor_alarm := FALSE;
   END_IF;

   (*Предупреждение. Авария ПЧ ДС*)
   IF "Sensors".DS_Invertor_alarm.Enable AND "Sensors".DS_invertor_mode.Value THEN
       "Alarms_and_warnings".Warning_DS_invertor_alarm := "Sensors".DS_Invertor_alarm.Value;
   ELSE
       "Alarms_and_warnings".Warning_DS_invertor_alarm := FALSE;
   END_IF;

   (*Предупреждение. ЗРГ в местном режиме управления*)
   "Alarms_and_warnings".Warning_ZRG_manual := NOT "Sensors".ZRG_avto.Value;

   (*Предупреждение. НАВ в местном режиме управления*)
   "Alarms_and_warnings".Warning_NAV_manual := NOT "Sensors".NAV_avto.Value;

   (*Предупреждение. НАД в местном режиме управления*)
   "Alarms_and_warnings".Warning_NAD_manual := NOT "Sensors".NAD_avto.Value;

   (*Предупреждение. ДВ в местном режиме управления*)
   "Alarms_and_warnings".Warning_DV_manual := "Sensors".DV_local_control.Value;

   (*Предупреждение. ДС в местном режиме управления*)
   "Alarms_and_warnings".Warning_DS_manual := "Sensors".DS_local_control.Value;

   (*Пламя запальника потухло*)
   "Timer".alarm_16_PT := T_CONV(INT_TO_DINT("Alarms_and_warnings".TIME_Warning_Not_flame_Igniter));
   IF "Alarms_and_warnings".Enable_Warning_Not_flame_Igniter THEN
       "Timer".alarm_16_IN := NOT "Sensors".Igniter_flame.Value;
       IF "Timer".alarm_16_Q THEN
           "Alarms_and_warnings".Warning_Not_flame_Igniter := TRUE;
       END_IF;
   ELSE
       "Timer".alarm_16_IN := FALSE;
       "Alarms_and_warnings".Warning_Not_flame_Igniter := FALSE;
   END_IF;

   (*ПЗК2 не открылся*)
   "Timer".alarm_17_PT := T_CONV(INT_TO_DINT("Alarms_and_warnings".TIME_Warning_PZK2_not_open) * 1000);
   IF "Alarms_and_warnings".Enable_Warning_PZK2_not_open THEN
       "Timer".alarm_17_IN := NOT "Sensors".PZK2_open.Value;
       IF "Timer".alarm_17_Q THEN
           "Alarms_and_warnings".Warning_PZK2_not_open := TRUE;
       END_IF;
   ELSE
       "Timer".alarm_17_IN := FALSE;
       "Alarms_and_warnings".Warning_PZK2_not_open := FALSE;
   END_IF;

   (*Понижение давления сетевой воды перед котлом*)
   IF "Sensors".P_water_before_boiler_min.Value OR ("Sensors".P_water_before_boiler.Value < "Alarms_and_warnings".SP_warning_L_P_water_before_boiler AND NOT "Alarms_and_warnings".Warning_sensor_P_water_before_boiler AND "Sensors".P_water_before_boiler.Enable) THEN
       "Alarms_and_warnings".Warning_P_water_before_boiler_min := TRUE;
   ELSE
       "Alarms_and_warnings".Warning_P_water_before_boiler_min := FALSE;
   END_IF;

   (*Повышение давления сетевой воды перед котлом*)
   IF "Sensors".P_water_before_boiler_max.Value OR ("Sensors".P_water_before_boiler.Value > "Alarms_and_warnings".SP_warning_H_P_water_before_boiler AND NOT "Alarms_and_warnings".Warning_sensor_P_water_before_boiler AND "Sensors".P_water_before_boiler.Enable) THEN
       "Alarms_and_warnings".Warning_P_water_before_boiler_max := TRUE;
   ELSE
       "Alarms_and_warnings".Warning_P_water_before_boiler_max := FALSE;
   END_IF;

   (*Понижение давления сетевой воды после котла*)
   IF "Sensors".P_water_after_boiler_min.Value OR ("Sensors".P_water_after_boiler.Value < "Alarms_and_warnings".SP_warning_L_P_water_after_boiler AND NOT "Alarms_and_warnings".Warning_sensor_P_water_after_boiler AND "Sensors".P_water_after_boiler.Enable) THEN
       "Alarms_and_warnings".Warning_P_water_after_boiler_min := TRUE;
   ELSE
       "Alarms_and_warnings".Warning_P_water_after_boiler_min := FALSE;
   END_IF;

   (*Повышение давления сетевой воды после котла*)
   IF "Sensors".P_water_after_boiler_max.Value OR ("Sensors".P_water_after_boiler.Value > "Alarms_and_warnings".SP_warning_H_P_water_after_boiler AND NOT "Alarms_and_warnings".Warning_sensor_P_water_after_boiler AND "Sensors".P_water_after_boiler.Enable) THEN
       "Alarms_and_warnings".Warning_P_water_after_boiler_max := TRUE;
   ELSE
       "Alarms_and_warnings".Warning_P_water_after_boiler_max := FALSE;
   END_IF;

   (*Повышение температуры сетевой воды после котла*)
   IF ("Sensors".T_water_after_boiler.Value > "Alarms_and_warnings".SP_warning_H_T_water_after_boiler AND NOT "Alarms_and_warnings".Warning_sensor_T_water_after_boiler AND "Sensors".T_water_after_boiler.Enable) THEN
       "Alarms_and_warnings".Warning_T_water_after_boiler_max := TRUE;
   ELSE
       "Alarms_and_warnings".Warning_T_water_after_boiler_max := FALSE;
   END_IF;

   (*Повышение расхода сетевой воды через котел*)
   IF "Sensors".Q_water_boiler_max.Value OR ("Sensors".Q_water_boiler.Value > "Alarms_and_warnings".SP_warning_H_Q_water_boiler AND "Sensors".Q_water_boiler.Enable) THEN
       "Alarms_and_warnings".Warning_Q_water_boiler_max := TRUE;
   ELSE
       "Alarms_and_warnings".Warning_Q_water_boiler_max := FALSE;
   END_IF;

   (*Понижение расхода сетевой воды через котел*)
   IF ("Sensors".Q_water_boiler.Value < "Alarms_and_warnings".SP_warning_L_Q_water_boiler AND "Sensors".Q_water_boiler.Enable) THEN
       "Alarms_and_warnings".Warning_Q_water_boiler_min := TRUE;
   ELSE
       "Alarms_and_warnings".Warning_Q_water_boiler_min := FALSE;
   END_IF;

   (*СО порог 1*)
   IF "Sensors".CO_1.Value THEN
       "Alarms_and_warnings".Warning_CO2_porog1 := TRUE;
   ELSE
       "Alarms_and_warnings".Warning_CO2_porog1 := FALSE;
   END_IF;

   (*Предупреждение. Неисправность датчика P газа перед горелкой*)
   IF "Sensors".P_gas_before_BG.Enable THEN
       "Alarms_and_warnings".Warning_sensor_P_gas_before_BG := "Sensors".P_gas_before_BG.Alarm_sensor;
   ELSE
       "Alarms_and_warnings".Warning_sensor_P_gas_before_BG := FALSE;
   END_IF;

   (*Предупреждение. Понижение разряжения в топке*)
   "Timer".warning_1_PT := T_CONV(INT_TO_DINT("Alarms_and_warnings".TIME_Alarm_dP_furnace_boiler_min) * 1000);
   IF "Technology".Regim = 3 AND ("Technology".Regim_ventilation_step = 23 OR "Technology".Regim_ventilation_step = 24) THEN
       "Timer".warning_1_IN := "Sensors".dP_furnace_boiler_min.Value OR ("Sensors".dP_furnace_boiler.Value > "Alarms_and_warnings".SP_alarm_L_dP_furnace_boiler AND NOT "Alarms_and_warnings".Warning_sensor_dP_furnace_boiler AND "Sensors".dP_furnace_boiler.Enable);
       IF "Timer".warning_1_Q THEN
           "Alarms_and_warnings".Warning_dP_furnace_boiler_min := TRUE;
       END_IF;
   ELSE
       "Timer".warning_1_IN := FALSE;
       "Alarms_and_warnings".Warning_dP_furnace_boiler_min := FALSE;
   END_IF;

   (*Предупреждение. Понижение давления воздуха перед горелкой *)
   "Timer".warning_2_PT := T_CONV(INT_TO_DINT("Alarms_and_warnings".TIME_Alarm_P_air_before_burner_min) * 1000);
   IF "Technology".Regim = 3 AND ("Technology".Regim_ventilation_step = 23 OR "Technology".Regim_ventilation_step = 24) THEN
       "Timer".warning_2_IN := "Sensors".P_air_before_burner_min.Value OR ("Sensors".P_air_burner.Value < "Alarms_and_warnings".SP_alarm_L_P_air_before_burner AND NOT "Alarms_and_warnings".Warning_sensor_P_air_burner AND "Sensors".P_air_burner.Enable);
       IF "Timer".warning_2_Q THEN
           "Alarms_and_warnings".Warning_P_air_before_burner_min := TRUE;
       END_IF;
   ELSE
       "Timer".warning_2_IN := FALSE;
       "Alarms_and_warnings".Warning_P_air_before_burner_min := FALSE;
   END_IF;

   (*ЗДГ не закрылась*)
   "Timer".warning_3_PT := T_CONV(INT_TO_DINT("Alarms_and_warnings".TIME_Warning_ZDG_not_close) * 1000);
   IF "Alarms_and_warnings".Enable_Warning_ZDG_not_close THEN
       "Timer".warning_3_IN := "Sensors".ZDG_no_close.Value;
       IF "Timer".warning_3_Q THEN
           "Alarms_and_warnings".Warning_ZDG_not_close := TRUE;
       END_IF;
   ELSE
       "Timer".warning_3_IN := FALSE;
   END_IF;

   (*Предупреждение. Имеется блокировка защиты *)
   IF "Protections".BLOCK_P_gas_before_BG_max OR
       "Protections".BLOCK_P_gas_before_BG_min OR
       "Protections".BLOCK_P_gas_before_burner_min OR
       "Protections".BLOCK_P_gas_before_burner_max OR
       "Protections".BLOCK_DS_off OR
       "Protections".BLOCK_DV_off OR
       "Protections".BLOCK_dP_in_furnance_min OR
       "Protections".BLOCK_P_air_before_burner_min OR
       "Protections".BLOCK_P_water_after_boiler_min OR
       "Protections".BLOCK_P_water_after_boiler_max OR
       "Protections".BLOCK_T_water_after_boiler_max OR
       "Protections".BLOCK_Q_water_boiler_min OR
       "Protections".BLOCK_Not_flame_burner OR
       "Protections".BLOCK_Alarm_stop_HMI OR
       "Protections".BLOCK_Alarm_stop_SCADA OR
       "Protections".BLOCK_CO2_porog2 OR
       "Protections".BLOCK_CH4 THEN
       "Alarms_and_warnings".Warning_protection_block := TRUE;
   ELSE
       "Alarms_and_warnings".Warning_protection_block := FALSE;
   END_IF;

   (*СБРОС аварий для журнала событий*)
   IF "Alarms_and_warnings".Reset_alarms THEN
       "HMI".Reset_alarms_Log := TRUE;
   END_IF;

   (*Сброс всех аварий и предупреждений*)
   IF "Alarms_and_warnings".Reset_alarms = TRUE OR
       "Sensors".Btn_Sound.Value THEN
       (*Повышение давления газа перед БГ*)
       IF NOT "Timer".alarm_1_Q THEN
           "Alarms_and_warnings".Alarm_P_gas_before_BG_max := FALSE;
       END_IF;
       (*Понижение давления газа перед БГ*)
       IF NOT "Timer".alarm_2_Q THEN
           "Alarms_and_warnings".Alarm_P_gas_before_BG_min := FALSE;
       END_IF;
       (*Понижение давления газа перед горелкой*)
       IF NOT "Timer".alarm_3_Q THEN
           "Alarms_and_warnings".Alarm_P_gas_before_burner_min := FALSE;
       END_IF;
       (*Повышение давления газа перед горелкой*)
       IF NOT "Timer".alarm_4_Q THEN
           "Alarms_and_warnings".Alarm_P_gas_before_burner_max := FALSE;
       END_IF;
       (*Отключение ДС*)
       IF NOT "Timer".alarm_5_Q THEN
           "Alarms_and_warnings".Alarm_DS_off := FALSE;
       END_IF;
       (*Отключение ДВ*)
       IF NOT "Timer".alarm_6_Q THEN
           "Alarms_and_warnings".Alarm_DV_off := FALSE;
       END_IF;
       (*Понижение разряжения в топке*)
       IF NOT "Timer".alarm_7_Q THEN
           "Alarms_and_warnings".Alarm_dP_furnace_boiler_min := FALSE;
       END_IF;
       (*Понижение давления воздуха перед горелкой *)
       IF NOT "Timer".alarm_8_Q THEN
           "Alarms_and_warnings".Alarm_P_air_before_burner_min := FALSE;
       END_IF;
       (*Понижение давления сетевой воды за котлом*)
       IF NOT "Timer".alarm_9_Q THEN
           "Alarms_and_warnings".Alarm_P_water_after_boiler_min := FALSE;
       END_IF;
       (*Повышение давления сетевой воды за котлом*)
       IF NOT "Timer".alarm_10_Q THEN
           "Alarms_and_warnings".Alarm_P_water_after_boiler_max := FALSE;
       END_IF;
       (*Повышение температуры сетевой воды за котлом*)
       IF NOT "Timer".alarm_11_Q THEN
           "Alarms_and_warnings".Alarm_T_water_after_boiler_max := FALSE;
       END_IF;
       (*Понижение расхода сетевой воды через котел*)
       IF NOT "Timer".alarm_12_Q THEN
           "Alarms_and_warnings".Alarm_Q_water_boiler_min := FALSE;
       END_IF;
       (*Невоспламенение или погасание факела горелки котла*)
       IF NOT "Timer".alarm_13_Q THEN
           "Alarms_and_warnings".Alarm_Not_flame_burner := FALSE;
       END_IF;
       "Alarms_and_warnings".Alarm_stop_HMI := FALSE;
       "Alarms_and_warnings".Alarm_stop_SCADA := FALSE;
       (*СО2 порог 2*)
       IF NOT "Timer".alarm_14_Q THEN
           "Alarms_and_warnings".Alarm_CO2_porog2 := FALSE;
       END_IF;
       (*CH4*)
       IF NOT "Timer".alarm_15_Q THEN
           "Alarms_and_warnings".Alarm_CH4 := FALSE;
       END_IF;
       //"Alarms_and_warnings".Warning_sensor_T_water_before_boiler := FALSE;
       //"Alarms_and_warnings".Warning_sensor_P_water_before_boiler := FALSE;
       //"Alarms_and_warnings".Warning_sensor_dP_water_boiler := FALSE;
       //"Alarms_and_warnings".Warning_sensor_T_water_after_boiler := FALSE;
       //"Alarms_and_warnings".Warning_sensor_P_water_after_boiler := FALSE;
       //"Alarms_and_warnings".Warning_sensor_dP_water_boiler_1 := FALSE;
       //"Alarms_and_warnings".Warning_sensor_P_water_before_boiler_1 := FALSE;
       //"Alarms_and_warnings".Warning_sensor_dP_gas_boiler := FALSE;
       //"Alarms_and_warnings".Warning_sensor_dP_furnace_boiler := FALSE;
       //"Alarms_and_warnings".Warning_sensor_P_gas_before_PZK1_and_PZK2 := FALSE;
       //"Alarms_and_warnings".Warning_sensor_P_gas_before_burner := FALSE;
       //"Alarms_and_warnings".Warning_sensor_P_air_burner := FALSE;
       //"Alarms_and_warnings".Warning_sensor_T_exhaust_gas := FALSE;
       //"Alarms_and_warnings".Warning_sensor_ZRG_position := FALSE;
       //"Alarms_and_warnings".Warning_sensor_NAV_position := FALSE;
       //"Alarms_and_warnings".Warning_sensor_NAD_position := FALSE;
       //"Alarms_and_warnings".Warning_sensor_DV_current_frequency := FALSE;
       //"Alarms_and_warnings".Warning_sensor_DS_current_frequency := FALSE;
       //"Alarms_and_warnings".Warning_ZDSV_before_boiler_limit_rotational_moment := FALSE;
       //"Alarms_and_warnings".Warning_ZDSV_after_boiler_limit_rotational_moment := FALSE;
       //"Alarms_and_warnings".Warning_сall_power_supply_сabinet := FALSE;
       //"Alarms_and_warnings".Warning_DV_need_on_QF_invertor := FALSE;
       //"Alarms_and_warnings".Warning_DV_need_on_QF_powergrid := FALSE;
       //"Alarms_and_warnings".Warning_DV_no_voltage := FALSE;
       //"Alarms_and_warnings".Warning_DS_need_on_QF_invertor := FALSE;
       //"Alarms_and_warnings".Warning_DS_need_on_QF_powergrid := FALSE;
       //"Alarms_and_warnings".Warning_DS_no_voltage := FALSE;
       //"Alarms_and_warnings".Warning_SHEU_no_voltage := FALSE;
       //"Alarms_and_warnings".Warning_power_PLC_from_UPS := FALSE;
       //"Alarms_and_warnings".Warning_UPS_Low_charge := FALSE;
       //"Alarms_and_warnings".Warning_ZRG_no_voltage := FALSE;
       //"Alarms_and_warnings".Warning_ZDG_no_voltage := FALSE;
       //"Alarms_and_warnings".Warning_NAV_no_voltage := FALSE;
       //"Alarms_and_warnings".Warning_NAD_no_voltage := FALSE;
       //"Alarms_and_warnings".Warning_ZDSV_before_boiler_no_voltage := FALSE;
       //"Alarms_and_warnings".Warning_ZDSV_after_boiler_no_voltage := FALSE;
       //"Alarms_and_warnings".Warning_DV_invertor_alarm := FALSE;
       //"Alarms_and_warnings".Warning_DS_invertor_alarm := FALSE;
       //"Alarms_and_warnings".Warning_ZRG_manual := FALSE;
       //"Alarms_and_warnings".Warning_NAV_manual := FALSE;
       //"Alarms_and_warnings".Warning_NAD_manual := FALSE;
       //"Alarms_and_warnings".Warning_DV_manual := FALSE;
       //"Alarms_and_warnings".Warning_DS_manual := FALSE;
       (*Пламя запальника потухло*)
       IF NOT "Timer".alarm_16_Q THEN
           "Alarms_and_warnings".Warning_Not_flame_Igniter := FALSE;
       END_IF;
       (*ПЗК2 не открылся*)
       IF NOT "Timer".alarm_17_Q THEN
           "Alarms_and_warnings".Warning_PZK2_not_open := FALSE;
       END_IF;
       //"Alarms_and_warnings".Warning_P_water_before_boiler_min := FALSE;
       //"Alarms_and_warnings".Warning_P_water_before_boiler_max := FALSE;
       //"Alarms_and_warnings".Warning_P_water_after_boiler_min := FALSE;
       //"Alarms_and_warnings".Warning_P_water_after_boiler_max := FALSE;
       //"Alarms_and_warnings".Warning_T_water_after_boiler_max := FALSE;
       //"Alarms_and_warnings".Warning_Q_water_boiler_max := FALSE;
       //"Alarms_and_warnings".Warning_Q_water_boiler_min := FALSE;
       //"Alarms_and_warnings".Warning_CO2_porog1 := FALSE;
       //"Alarms_and_warnings".Warning_sensor_P_gas_before_BG := FALSE;
       (*Предупреждение. Понижение разряжения в топке*)
       IF NOT "Timer".warning_1_Q THEN
           "Alarms_and_warnings".Warning_dP_furnace_boiler_min := FALSE;
       END_IF;
       (*Предупреждение. Понижение давления воздуха перед горелкой *)
       IF NOT "Timer".warning_2_Q THEN
           "Alarms_and_warnings".Warning_P_air_before_burner_min := FALSE;
       END_IF;
       (*ЗДГ не закрылась*)
       IF NOT "Timer".warning_3_Q THEN
           "Alarms_and_warnings".Warning_ZDG_not_close := FALSE;
       END_IF;
       //"Alarms_and_warnings".Warning_protection_block := FALSE;
       "Alarms_and_warnings".Reset_alarms := FALSE;
   END_IF;

   (*Формирование обобщенного признака аварии*)
   "Alarms_and_warnings".Global_alarm := "Alarms_and_warnings".Alarm_P_gas_before_BG_max OR
   "Alarms_and_warnings".Alarm_P_gas_before_BG_min OR
   "Alarms_and_warnings".Alarm_P_gas_before_burner_min OR
   "Alarms_and_warnings".Alarm_P_gas_before_burner_max OR
   "Alarms_and_warnings".Alarm_DS_off OR
   "Alarms_and_warnings".Alarm_DV_off OR
   "Alarms_and_warnings".Alarm_dP_furnace_boiler_min OR
   "Alarms_and_warnings".Alarm_P_air_before_burner_min OR
   "Alarms_and_warnings".Alarm_P_water_after_boiler_min OR
   "Alarms_and_warnings".Alarm_P_water_after_boiler_max OR
   "Alarms_and_warnings".Alarm_T_water_after_boiler_max OR
   "Alarms_and_warnings".Alarm_Q_water_boiler_min OR
   "Alarms_and_warnings".Alarm_Not_flame_burner OR
   "Alarms_and_warnings".Alarm_stop_HMI OR
   "Alarms_and_warnings".Alarm_stop_SCADA OR
   "Alarms_and_warnings".Alarm_CO2_porog2 OR
   "Alarms_and_warnings".Alarm_CH4;

   (*ловим передний фронт аварий*)                                        
   "R_TRIG_DB_11"(CLK := "Alarms_and_warnings".Alarm_P_gas_before_BG_max,
                  Q => "FRONT_Alarm_1");
   "R_TRIG_DB_12"(CLK := "Alarms_and_warnings".Alarm_P_gas_before_BG_min,
                  Q => "FRONT_Alarm_2");
   "R_TRIG_DB_13"(CLK := "Alarms_and_warnings".Alarm_P_gas_before_burner_min,
                  Q => "FRONT_Alarm_3");
   "R_TRIG_DB_14"(CLK := "Alarms_and_warnings".Alarm_P_gas_before_burner_max,
                  Q => "FRONT_Alarm_4");
   "R_TRIG_DB_15"(CLK := "Alarms_and_warnings".Alarm_DS_off,
                  Q => "FRONT_Alarm_5");
   "R_TRIG_DB_16"(CLK := "Alarms_and_warnings".Alarm_DV_off,
                  Q => "FRONT_Alarm_6");
   "R_TRIG_DB_17"(CLK := "Alarms_and_warnings".Alarm_dP_furnace_boiler_min,
                  Q => "FRONT_Alarm_7");
   "R_TRIG_DB_18"(CLK := "Alarms_and_warnings".Alarm_P_air_before_burner_min,
                  Q => "FRONT_Alarm_8");
   "R_TRIG_DB_19"(CLK := "Alarms_and_warnings".Alarm_P_water_after_boiler_min,
                  Q => "FRONT_Alarm_9");
   "R_TRIG_DB_20"(CLK := "Alarms_and_warnings".Alarm_P_water_after_boiler_max,
                  Q => "FRONT_Alarm_10");
   "R_TRIG_DB_21"(CLK := "Alarms_and_warnings".Alarm_T_water_after_boiler_max,
                  Q => "FRONT_Alarm_11");
   "R_TRIG_DB_22"(CLK := "Alarms_and_warnings".Alarm_Q_water_boiler_min,
                  Q => "FRONT_Alarm_12");
   "R_TRIG_DB_23"(CLK := "Alarms_and_warnings".Alarm_Not_flame_burner,
                  Q => "FRONT_Alarm_13");
   "R_TRIG_DB_24"(CLK := "Alarms_and_warnings".Alarm_stop_HMI,
                  Q => "FRONT_Alarm_14");
   "R_TRIG_DB_25"(CLK := "Alarms_and_warnings".Alarm_stop_SCADA,
                  Q => "FRONT_Alarm_15");
   "R_TRIG_DB_26"(CLK := "Alarms_and_warnings".Alarm_CO2_porog2,
                  Q => "FRONT_Alarm_16");
   "R_TRIG_DB_27"(CLK := "Alarms_and_warnings".Alarm_CH4,
                  Q => "FRONT_Alarm_17");

   (*Управление звуковой сигнализацией*)
   "Timer".test_sound_PT := T#2s;
   "Timer".test_sound_IN := "Sensors".Btn_Sound.Value;
   IF "FRONT_Alarm_1" OR
       "FRONT_Alarm_2" OR
       "FRONT_Alarm_3" OR
       "FRONT_Alarm_4" OR
       "FRONT_Alarm_5" OR
       "FRONT_Alarm_6" OR
       "FRONT_Alarm_7" OR
       "FRONT_Alarm_8" OR
       "FRONT_Alarm_9" OR
       "FRONT_Alarm_10" OR
       "FRONT_Alarm_11" OR
       "FRONT_Alarm_12" OR
       "FRONT_Alarm_13" OR
       "FRONT_Alarm_14" OR
       "FRONT_Alarm_15" OR
       "FRONT_Alarm_16" OR
       "FRONT_Alarm_17" OR
       "Timer".test_sound_Q THEN
       "Sensors".control_alarm_signal.Value := TRUE;
   ELSE
       //отключение звуковой сигнализации
       IF (NOT "Alarms_and_warnings".Global_alarm AND NOT "Timer".test_sound_Q) OR "FRONT_Btn_reset_sound_HMI" THEN
           "Sensors".control_alarm_signal.Value := FALSE;
       END_IF;
   END_IF;
END_FUNCTION

FUNCTION "Protection" : Void   // FC8, SCL
{ S7_Optimized_Access := 'TRUE' }
VERSION : 0.1
BEGIN
   (*Принудительный сброс блокировок защит*)
   (* (*Повышение давления газа перед БГ*)
   "TON_protection_1_DB".TON(IN := "Protections".BLOCK_P_gas_before_BG_max,
                             PT := T#15m,
                             Q => "Timer".protection_1_Q);
   IF "Timer".protection_1_Q THEN
       "Protections".BLOCK_P_gas_before_BG_max := FALSE;
   END_IF; *)
   (* (*Понижение давления газа перед БГ*)
   "TON_protection_2_DB".TON(IN := "Protections".BLOCK_P_gas_before_BG_min,
                             PT := T#15m,
                             Q => "Timer".protection_2_Q);
   IF "Timer".protection_2_Q THEN
       "Protections".BLOCK_P_gas_before_BG_min := FALSE;
   END_IF; *)
   (* (*Понижение давления газа перед горелкой*)
   "TON_protection_3_DB".TON(IN :="Protections".BLOCK_P_gas_before_burner_min,
                             PT := T#15m,
                             Q => "Timer".protection_3_Q);
   IF "Timer".protection_3_Q THEN
       "Protections".BLOCK_P_gas_before_burner_min := FALSE;
   END_IF; *)
   (* (*Повышение давления газа перед горелкой*)
   "TON_protection_4_DB".TON(IN :="Protections".BLOCK_P_gas_before_burner_max,
                             PT := T#15m,
                             Q => "Timer".protection_4_Q);
   IF "Timer".protection_4_Q THEN
       "Protections".BLOCK_P_gas_before_burner_max := FALSE;
   END_IF; *)
   (* (*Отключение ДС*)
   "TON_protection_5_DB".TON(IN :="Protections".BLOCK_DS_off,
                             PT := T#15m,
                             Q => "Timer".protection_5_Q);
   IF "Timer".protection_5_Q THEN
       "Protections".BLOCK_DS_off := FALSE;
   END_IF; *)
   (* (*Отключение ДВ*)
   "TON_protection_6_DB".TON(IN :="Protections".BLOCK_DV_off,
                             PT := T#15m,
                             Q => "Timer".protection_6_Q);
   IF "Timer".protection_6_Q THEN
       "Protections".BLOCK_DV_off:= FALSE;
   END_IF; *)
   (* (*Понижение разряжения в топке*)
   "TON_protection_7_DB".TON(IN :="Protections".BLOCK_dP_in_furnance_min,
                             PT := T#15m,
                             Q => "Timer".protection_7_Q);
   IF "Timer".protection_7_Q THEN
       "Protections".BLOCK_dP_in_furnance_min:= FALSE;
   END_IF; *)
   (* (*Понижение давления воздуха перед горелкой*)
   "TON_protection_8_DB".TON(IN :="Protections".BLOCK_P_air_before_burner_min,
                             PT := T#15m,
                             Q => "Timer".protection_8_Q);
   IF "Timer".protection_8_Q THEN
       "Protections".BLOCK_P_air_before_burner_min:= FALSE;
   END_IF; *)
   (* (*Понижение давления сетевой воды за котлом*)
   "TON_protection_9_DB".TON(IN :="Protections".BLOCK_P_water_after_boiler_min,
                             PT := T#15m,
                             Q => "Timer".protection_9_Q);
   IF "Timer".protection_9_Q THEN
       "Protections".BLOCK_P_water_after_boiler_min:= FALSE;
   END_IF; *)
   (* (*Повышение давления сетевой воды за котлом*)
   "TON_protection_10_DB".TON(IN :="Protections".BLOCK_P_water_after_boiler_max,
                             PT := T#15m,
                             Q => "Timer".protection_10_Q);
   IF "Timer".protection_10_Q THEN
       "Protections".BLOCK_P_water_after_boiler_max:= FALSE;
   END_IF; *)
   (* (*Повышение температуры сетевой воды за котлом*)
   "TON_protection_11_DB".TON(IN :="Protections".BLOCK_T_water_after_boiler_max,
                             PT := T#15m,
                             Q => "Timer".protection_11_Q);
   IF "Timer".protection_11_Q THEN
       "Protections".BLOCK_T_water_after_boiler_max:= FALSE;
   END_IF; *)
   (* (*Понижение расхода сетевой воды через котел*)
   "TON_protection_12_DB".TON(IN :="Protections".BLOCK_Q_water_boiler_min,
                             PT := T#15m,
                             Q => "Timer".protection_12_Q);
   IF "Timer".protection_12_Q THEN
       "Protections".BLOCK_Q_water_boiler_min:= FALSE;
   END_IF; *)
   (*Невоспламенение или погасание факела горелки котла*)
   "TON_protection_13_DB".TON(IN :="Protections".BLOCK_Not_flame_burner,
                             PT := T#5m,
                             Q => "Timer".protection_13_Q);
   IF "Timer".protection_13_Q THEN
       "Protections".BLOCK_Not_flame_burner:= FALSE;
   END_IF;
   (* (*Нажата кнопка аварийного останова на панели операторора*)
   "TON_protection_14_DB".TON(IN :="Protections".BLOCK_Alarm_stop_HMI,
                             PT := T#15m,
                             Q => "Timer".protection_14_Q);
   IF "Timer".protection_14_Q THEN
       "Protections".BLOCK_Alarm_stop_HMI:= FALSE;
   END_IF; *)
   (* (*Нажата кнопка аварийного останова на SCADA*)
   "TON_protection_15_DB".TON(IN :="Protections".BLOCK_Alarm_stop_SCADA,
                             PT := T#15m,
                             Q => "Timer".protection_15_Q);
   IF "Timer".protection_15_Q THEN
       "Protections".BLOCK_Alarm_stop_SCADA:= FALSE;
   END_IF; *)
   (* (*СО2 порог 2*)
   "TON_protection_16_DB".TON(IN :="Protections".BLOCK_CO2_porog2,
                             PT := T#15m,
                             Q => "Timer".protection_16_Q);
   IF "Timer".protection_16_Q THEN
       "Protections".BLOCK_CO2_porog2:= FALSE;
   END_IF; *)
   (* (*CH4*)
   "TON_protection_17_DB".TON(IN :="Protections".BLOCK_CH4,
                             PT := T#15m,
                             Q => "Timer".protection_17_Q);
   IF "Timer".protection_17_Q THEN
       "Protections".BLOCK_CH4:= FALSE;
   END_IF; *)

   (*формирование обобщенного признака сработки защиты*)
   IF "Protections".P_gas_before_BG_max OR
       "Protections".P_gas_before_BG_min OR
       "Protections".P_gas_before_burner_min OR
       "Protections".P_gas_before_burner_max OR
       "Protections".DS_off OR
       "Protections".DV_off OR
       "Protections".dP_in_furnance_min OR
       "Protections".P_air_before_burner_min OR
       "Protections".P_water_after_boiler_min OR
       "Protections".P_water_after_boiler_max OR
       "Protections".T_water_after_boiler_max OR
       "Protections".Q_water_boiler_min OR
       "Protections".Not_flame_burner OR
       "Protections".Alarm_stop_HMI OR
       "Protections".Alarm_stop_SCADA OR
       "Protections".CO2_porog2 OR
       "Protections".CH4 THEN
       "Protections".Global := TRUE;
   ELSE
       "Protections".Global := FALSE;
   END_IF;
END_FUNCTION

FUNCTION "Select_regim" : Void   // FC9, SCL
{ S7_Optimized_Access := 'TRUE' }
VERSION : 0.1
BEGIN
   (*Выбор режима работы*)
   (*  1-ОТКЛ
       2-ПРОВЕРКА
       3-ВЕНТИЛЯЦИЯ
       4-ОПРЕССОВКА
       5-РОЗЖИГ
       6-ВЫХОД НА МИНИМАЛЬНУЮ МОЩНОСТЬ
       7-ПРОГРЕВ
       8-РАБОТА
       9-ЭКСТРЕННЫЙ ОСТАНОВ
       10-АВАРИЙНЫЙ ОСТАНОВ
       11-ПЛАНОВЫЙ ОСТАНОВ
       12-ПОСТОСТАНОВОЧНАЯ ОПРЕССОВКА
       13-УКОРОЧЕННАЯ ВЕНТИЛЯЦИЯ
       14-ТЕСТОВАЯ ОПРЕССОВКА
       15-ТЕСТОВЫЙ РОЗЖИГ*)
   IF "Technology".Regim <= 0 OR "Technology".Regim >= 16 THEN
       "Technology".Regim := 1;
   END_IF;

   (*Экстренный останов*)
   IF "Sensors".Btn_STOP.Value THEN
       "Technology".Regim := 9;
   END_IF;

   (*Аварийный останов*)
   IF "Protections".Global THEN
       "Technology".Regim := 10;
   END_IF;

   (*Плановый останов*)
   IF ("FRONT_Btn_Normal_stop_HMI" OR "FRONT_Btn_Normal_stop_SCADA") AND "Technology".Regim <> 1 AND
       "Technology".Regim <> 10 AND
       "Technology".Regim <> 12 THEN
       "Technology".Regim := 11;
   END_IF;

   (* IF ("FRONT_Btn_Normal_stop_HMI" OR "FRONT_Btn_Normal_stop_SCADA") THEN
       "Technology".need_plan_stop := TRUE;
   END_IF;
   IF "Technology".need_plan_stop THEN
       IF  //если текущий режим ВЕНТИЛЯЦИЯ
           "Technology".Regim = 3 THEN
           IF //и наличие условия что вентиляция проведена или в режиме розжига ПЗК2 не открывался
               "Technology".Ventilation_conducted OR NOT "Technology".transition_ignition THEN
               //снимаем защиту Повышение давления газа перед БГ
               "Alarms_and_warnings".Enable_Alarm_P_gas_before_BG_max := FALSE;
               //снимаем защиту Понижение давления газа перед БГ
               "Alarms_and_warnings".Enable_Alarm_P_gas_before_BG_min := FALSE;
               //снимаем защиту Понижение давления газа перед горелкой
               "Alarms_and_warnings".Enable_Alarm_P_gas_before_burner_min := FALSE;
               //снимаем защиту Повышение давления газа перед горелкой
               "Alarms_and_warnings".Enable_Alarm_P_gas_before_burner_max := FALSE;
               //снимаем защиту Отключение ДС
               "Alarms_and_warnings".Enable_Alarm_DS_off := FALSE;
               //снимаем защиту Отключение ДВ
               "Alarms_and_warnings".Enable_Alarm_DV_off := FALSE;
               //снимаем защиту Понижение давления воздуха перед горелкой
               "Alarms_and_warnings".Enable_Alarm_P_air_before_burner_min := FALSE;
               //снимаем защиту Понижение разряжения в топке
               "Alarms_and_warnings".Enable_Alarm_dP_furnace_boiler_min := FALSE;
               //снимаем защиту Невоспламенение или погасание факела горелки котла
               "Alarms_and_warnings".Enable_Alarm_Not_flame_burner := FALSE;
               //все клапана переводим в исходное состояние
               "Control_PZK1".Mode := TRUE;    //закрываем ПЗК1
               "Control_PZK1".Avto_open := FALSE;
               "Control_PZK2".Mode := TRUE;    //закрываем ПЗК2
               "Control_PZK2".Avto_open := FALSE;
               "Control_KO".Mode := TRUE;  //закрываем КО
               "Control_KO".Avto_open := FALSE;
               "Control_KZ".Mode := TRUE;  //закрываем КЗ
               "Control_KZ".Avto_open := FALSE;
               "Control_KB".Mode := TRUE;  //открываем КБ
               "Control_KB".Avto_close := FALSE;
               "Control_IVN".Mode := TRUE; //отключаем ИВН
               "Control_IVN".Avto_on := FALSE;
           (* "Control_ZDG".Mode := TRUE; //закрываем ЗДГ
           "Control_ZDG".Avto_open := FALSE;
           "Control_ZDG".Avto_stop := FALSE;
           "Control_ZDG".Avto_close := TRUE; *)
               "Control_DV".Mode := TRUE;  //отключаем ДВ
               //"Control_DV".Mode_from_PLC := TRUE;
               "Control_DV".Avto_Start := FALSE;
               "Control_DV".Avto_Stop := TRUE;
               "Control_DS".Mode := TRUE;  //отключаем ДС
               //"Control_DS".Mode_from_PLC := TRUE;
               "Control_DS".Avto_Start := FALSE;
               "Control_DS".Avto_Stop := TRUE;
               IF  NOT "Sensors".PZK1_open.Value AND
                   NOT "Sensors".PZK2_open.Value AND
                   NOT "Sensors".PZK2_not_close.Value AND
                   NOT "Sensors".KO_open.Value AND
                   NOT "Sensors".KZ_open.Value AND
                   NOT "Sensors".KB_close.Value AND
                   NOT "Sensors".IVN_control_on.Value AND
                   NOT "Sensors".DV_invertor_on.Value AND
                   NOT "Sensors".DV_powergrid_on.Value AND
                   NOT "Sensors".DS_invertor_on.Value AND
                   NOT "Sensors".DS_powergrid_on.Value THEN
                   //переход на режим ОТКЛ
                   "Technology".Regim := 1;
                   "Technology".need_plan_stop := FALSE;
               END_IF;
           ELSE
               //переход на режим ПЛАНОВЫЙ ОСТАНОВ
               "Technology".Regim := 11;
               //на шаг 2
               "Technology".Regim_plan_stop_step := 2;
               //снимаем защиту Понижение давления газа перед горелкой
               "Alarms_and_warnings".Enable_Alarm_P_gas_before_burner_min := FALSE;
               //снимаем защиту Повышение давления газа перед горелкой
               "Alarms_and_warnings".Enable_Alarm_P_gas_before_burner_max := FALSE;
               "Technology".need_plan_stop := FALSE;
           END_IF;
       END_IF;

       IF  //если текущий режим ОПРЕССОВКА
           "Technology".Regim = 4 THEN
           //снимаем защиту Повышение давления газа перед БГ
           "Alarms_and_warnings".Enable_Alarm_P_gas_before_BG_max := FALSE;
           //снимаем защиту Понижение давления газа перед БГ
           "Alarms_and_warnings".Enable_Alarm_P_gas_before_BG_min := FALSE;
           //снимаем защиту Понижение давления газа перед горелкой
           "Alarms_and_warnings".Enable_Alarm_P_gas_before_burner_min := FALSE;
           //снимаем защиту Повышение давления газа перед горелкой
           "Alarms_and_warnings".Enable_Alarm_P_gas_before_burner_max := FALSE;
           //снимаем защиту Отключение ДС
           "Alarms_and_warnings".Enable_Alarm_DS_off := FALSE;
           //снимаем защиту Отключение ДВ
           "Alarms_and_warnings".Enable_Alarm_DV_off := FALSE;
           //снимаем защиту Понижение давления воздуха перед горелкой
           "Alarms_and_warnings".Enable_Alarm_P_air_before_burner_min := FALSE;
           //снимаем защиту Понижение разряжения в топке
           "Alarms_and_warnings".Enable_Alarm_dP_furnace_boiler_min := FALSE;
           //снимаем защиту Невоспламенение или погасание факела горелки котла
           "Alarms_and_warnings".Enable_Alarm_Not_flame_burner := FALSE;
           //все клапана переводим в исходное состояние
           "Control_PZK1".Mode := TRUE;    //закрываем ПЗК1
           "Control_PZK1".Avto_open := FALSE;
           "Control_PZK2".Mode := TRUE;    //закрываем ПЗК2
           "Control_PZK2".Avto_open := FALSE;
           "Control_KO".Mode := TRUE;  //закрываем КО
           "Control_KO".Avto_open := FALSE;
           "Control_KZ".Mode := TRUE;  //закрываем КЗ
           "Control_KZ".Avto_open := FALSE;
           "Control_KB".Mode := TRUE;  //открываем КБ
           "Control_KB".Avto_close := FALSE;
           "Control_IVN".Mode := TRUE; //отключаем ИВН
           "Control_IVN".Avto_on := FALSE;
           (* "Control_ZDG".Mode := TRUE; //закрываем ЗДГ
           "Control_ZDG".Avto_open := FALSE;
           "Control_ZDG".Avto_stop := FALSE;
           "Control_ZDG".Avto_close := TRUE; *)
           "Control_DV".Mode := TRUE;  //отключаем ДВ
           //"Control_DV".Mode_from_PLC := TRUE;
           "Control_DV".Avto_Start := FALSE;
           "Control_DV".Avto_Stop := TRUE;
           "Control_DS".Mode := TRUE;  //отключаем ДС
           //"Control_DS".Mode_from_PLC := TRUE;
           "Control_DS".Avto_Start := FALSE;
           "Control_DS".Avto_Stop := TRUE;
           IF NOT "Sensors".PZK1_open.Value AND
               NOT "Sensors".PZK2_open.Value AND
               NOT "Sensors".PZK2_not_close.Value AND
               NOT "Sensors".KO_open.Value AND
               NOT "Sensors".KZ_open.Value AND
               NOT "Sensors".KB_close.Value AND
               NOT "Sensors".IVN_control_on.Value AND
               NOT "Sensors".DV_invertor_on.Value AND
               NOT "Sensors".DV_powergrid_on.Value AND
               NOT "Sensors".DS_invertor_on.Value AND
               NOT "Sensors".DS_powergrid_on.Value THEN
               //переход на режим ОТКЛ
               "Technology".Regim := 1;
               "Technology".need_plan_stop := FALSE;
           END_IF;
       END_IF;

       IF  //если текущий режим РОЗЖИГ
           "Technology".Regim = 5 THEN
           IF //и наличие условия что вентиляция проведена или в режиме розжига ПЗК2 не открывался
               "Technology".Ventilation_conducted OR NOT "Technology".transition_ignition THEN
               //снимаем защиту Повышение давления газа перед БГ
               "Alarms_and_warnings".Enable_Alarm_P_gas_before_BG_max := FALSE;
               //снимаем защиту Понижение давления газа перед БГ
               "Alarms_and_warnings".Enable_Alarm_P_gas_before_BG_min := FALSE;
               //снимаем защиту Понижение давления газа перед горелкой
               "Alarms_and_warnings".Enable_Alarm_P_gas_before_burner_min := FALSE;
               //снимаем защиту Повышение давления газа перед горелкой
               "Alarms_and_warnings".Enable_Alarm_P_gas_before_burner_max := FALSE;
               //снимаем защиту Отключение ДС
               "Alarms_and_warnings".Enable_Alarm_DS_off := FALSE;
               //снимаем защиту Отключение ДВ
               "Alarms_and_warnings".Enable_Alarm_DV_off := FALSE;
               //снимаем защиту Понижение давления воздуха перед горелкой
               "Alarms_and_warnings".Enable_Alarm_P_air_before_burner_min := FALSE;
               //снимаем защиту Понижение разряжения в топке
               "Alarms_and_warnings".Enable_Alarm_dP_furnace_boiler_min := FALSE;
               //снимаем защиту Невоспламенение или погасание факела горелки котла
               "Alarms_and_warnings".Enable_Alarm_Not_flame_burner := FALSE;
               //все клапана переводим в исходное состояние
               "Control_PZK1".Mode := TRUE;    //закрываем ПЗК1
               "Control_PZK1".Avto_open := FALSE;
               "Control_PZK2".Mode := TRUE;    //закрываем ПЗК2
               "Control_PZK2".Avto_open := FALSE;
               "Control_KO".Mode := TRUE;  //закрываем КО
               "Control_KO".Avto_open := FALSE;
               "Control_KZ".Mode := TRUE;  //закрываем КЗ
               "Control_KZ".Avto_open := FALSE;
               "Control_KB".Mode := TRUE;  //открываем КБ
               "Control_KB".Avto_close := FALSE;
               "Control_IVN".Mode := TRUE; //отключаем ИВН
               "Control_IVN".Avto_on := FALSE;
               (* "Control_ZDG".Mode := TRUE; //закрываем ЗДГ
               "Control_ZDG".Avto_open := FALSE;
               "Control_ZDG".Avto_stop := FALSE;
               "Control_ZDG".Avto_close := TRUE; *)
               "Control_DV".Mode := TRUE;  //отключаем ДВ
               //"Control_DV".Mode_from_PLC := TRUE;
               "Control_DV".Avto_Start := FALSE;
               "Control_DV".Avto_Stop := TRUE;
               "Control_DS".Mode := TRUE;  //отключаем ДС
               //"Control_DS".Mode_from_PLC := TRUE;
               "Control_DS".Avto_Start := FALSE;
               "Control_DS".Avto_Stop := TRUE;
               IF NOT "Sensors".PZK1_open.Value AND
                   NOT "Sensors".PZK2_open.Value AND
                   NOT "Sensors".PZK2_not_close.Value AND
                   NOT "Sensors".KO_open.Value AND
                   NOT "Sensors".KZ_open.Value AND
                   NOT "Sensors".KB_close.Value AND
                   NOT "Sensors".IVN_control_on.Value AND
                   NOT "Sensors".DV_invertor_on.Value AND
                   NOT "Sensors".DV_powergrid_on.Value AND
                   NOT "Sensors".DS_invertor_on.Value AND
                   NOT "Sensors".DS_powergrid_on.Value THEN
                   //переход на режим ОТКЛ
                   "Technology".Regim := 1;
                   "Technology".need_plan_stop := FALSE;
               END_IF;
           ELSE
               //переход на режим ПЛАНОВЫЙ ОСТАНОВ
               "Technology".Regim := 11;
               //на шаг 2
               "Technology".Regim_plan_stop_step := 2;
               //снимаем защиту Понижение давления газа перед горелкой
               "Alarms_and_warnings".Enable_Alarm_P_gas_before_burner_min := FALSE;
               //снимаем защиту Повышение давления газа перед горелкой
               "Alarms_and_warnings".Enable_Alarm_P_gas_before_burner_max := FALSE;
               "Technology".need_plan_stop := FALSE;
           END_IF;
       END_IF;

       IF //если текущий режим
           "Technology".Regim = 6 OR
           "Technology".Regim = 7 OR
           "Technology".Regim = 8 THEN
           "Technology".Regim := 11;
           "Technology".need_plan_stop := FALSE;
       END_IF;
   END_IF; *)

   (*сброс признака провентилированности топки*)
   IF "Sensors".PZK2_not_close.Value OR
       ((NOT "Sensors".DS_invertor_on.Value AND NOT "Sensors".DS_powergrid_on.Value) OR (NOT "Sensors".DV_invertor_on.Value AND NOT "Sensors".DV_powergrid_on.Value)) THEN
       "Technology".Ventilation_conducted := FALSE;
   END_IF;

   (*был переход в режим РОЗЖИГ и открытие ПЗК2*)
   IF "Technology".Ventilation_conducted THEN
       "Technology".transition_ignition := FALSE;
   END_IF;
   IF "Technology".Regim = 5 AND "Sensors".PZK2_not_close.Value THEN
       "Technology".transition_ignition := TRUE;
   END_IF;

   (*если текущий режим не ОТКЛ и не РУЧНОЙ РОЗЖИГ, то ИМ по газу принудительно переводим в автоматический режим *)
   IF "Technology".Regim = 1 OR
       ("Technology".Regim = 5 AND "Technology".Regim_ignition_step =19) THEN
       ;
   ELSE
       (*КБ*)
       "Control_KB".Mode := TRUE;
       (*KO*)
       "Control_KO".Mode := TRUE;
       (*КЗ*)
       "Control_KZ".Mode := TRUE;
       (*ПЗК1*)
       "Control_PZK1".Mode := TRUE;
       (*ПЗК2*)
       "Control_PZK2".Mode := TRUE;
       (*ЗДГ*)
       //"Control_ZDG".Mode := TRUE;
       (*ИВН*)
       "Control_IVN".Mode := TRUE;
   END_IF;

   (*сброс признака тестовой опрессовки, если текущий режим не вентиляция и не опрессовка*)
   IF "Technology".Regim <> 3 AND "Technology".Regim <> 4 THEN
       "Technology".Test_press_run := FALSE;
       "Message".TEST_PRESS_ok := FALSE;   //сброс сообщения об успешном прохождении тестовой опрессовки
   END_IF;

   (*Взведение и снятие защит нажатию кнопок аварийного останова*)
   IF "Technology".Regim = 2 OR
       "Technology".Regim = 3 OR
       "Technology".Regim = 4 OR
       "Technology".Regim = 5 OR
       "Technology".Regim = 6 OR
       "Technology".Regim = 7 OR
       "Technology".Regim = 8 OR
       "Technology".Regim = 11 THEN
       //взводим защиту Нажата кнопка аварийного останова на панели оператора
       "Alarms_and_warnings".Enable_Alarm_stop_HMI := TRUE;
       //взводим защиту Нажата кнопка аварийного останова на SCADA
       "Alarms_and_warnings".Enable_Alarm_stop_SCADA := TRUE;
   ELSE
       //снимаем защиту Нажата кнопка аварийного останова на панели оператора
       "Alarms_and_warnings".Enable_Alarm_stop_HMI := FALSE;
       //снимаем защиту Нажата кнопка аварийного останова на SCADA
       "Alarms_and_warnings".Enable_Alarm_stop_SCADA := FALSE;
   END_IF;

   (*Аварийные сообщения по загазованности (не являются защитами)*)
   //СО2 порог 2
   "Alarms_and_warnings".Enable_Alarm_CO2_porog2 := TRUE;
   //CH4
   "Alarms_and_warnings".Enable_Alarm_CH4 := TRUE;

   IF "Technology".SP_T_water_after_boiler < 40.0 THEN
       "Technology".SP_T_water_after_boiler := 40.0;
   END_IF;
   IF "Technology".SP_T_water_after_boiler > 120.0 THEN
       "Technology".SP_T_water_after_boiler := 120.0;
   END_IF;
END_FUNCTION

